	ARrStnFilterPressurePV 								: ARRAY [1..iStnQty] OF REAL;
	ARbStnFilterPressure1stLimitAlarm					: ARRAY [1..iStnQty] OF BOOL;
	ARbStnFilterPressure2ndLimitAlarm					: ARRAY [1..iStnQty] OF BOOL;

	ARbStnFilterPressureLowAlarm						: ARRAY [1..iStnQty] OF BOOL;
	ARbStnFilterPressureHighAlarm						: ARRAY [1..iStnQty] OF BOOL;
	
	ARrIncFilterPressurePV 								: ARRAY [1..iStnQty] OF REAL;
	ARbIncFilterPressure1stLimitAlarm					: ARRAY [1..iStnQty] OF BOOL;
	ARbIncFilterPressure2ndLimitAlarm					: ARRAY [1..iStnQty] OF BOOL;

(* xxxxxxxxxxxxxxxxxxxxxxxxxxxxxxxx Flow Switch Cltr xxxxxxxxxxxxxxxxxxxxxxxxxxxxxxxx*)
(*========================================================================*)

	ARrStnFlowSwitchPV 									: ARRAY [1..iStnQty] OF REAL;
	ARbStnFlowSwitch1stLimitAlarm						: ARRAY [1..iStnQty] OF BOOL;
	ARbStnFlowSwitch2ndLimitAlarm						: ARRAY [1..iStnQty] OF BOOL;

	ARrIncFlowSwitchPV 									: ARRAY [1..iStnQty] OF REAL;
	ARbIncFlowSwitch1stLimitAlarm						: ARRAY [1..iStnQty] OF BOOL;
	ARbIncFlowSwitch2ndLimitAlarm						: ARRAY [1..iStnQty] OF BOOL;

(* xxxxxxxxxxxxxxxxxxxxxxxxxxxxxxxx Compress Air Cltr xxxxxxxxxxxxxxxxxxxxxxxxxxxxxxxx*)
(*========================================================================*)

	ARrStnCompressAirPV 								: ARRAY [1..iStnQty] OF REAL;
	ARbStnCompressAir1stLimitAlarm						: ARRAY [1..iStnQty] OF BOOL;
	ARbStnCompressAir2ndLimitAlarm						: ARRAY [1..iStnQty] OF BOOL;

	ARrIncCompressAirPV 								: ARRAY [1..iStnQty] OF REAL;
	ARbIncCompressAir1stLimitAlarm						: ARRAY [1..iStnQty] OF BOOL;
	ARbIncCompressAir2ndLimitAlarm						: ARRAY [1..iStnQty] OF BOOL;

(* xxxxxxxxxxxxxxxxxxxxxxxxxxxxxx Weber Ultrasonic Cltr xxxxxxxxxxxxxxxxxxxxxxxxxxxxxx*)
(*========================================================================*)

	bWeberFbErrorReset 									: BOOL;

	ARbUSFSel1OnOff 									: ARRAY [1..iUSGeneratorQty] OF BOOL;
	ARbUSFSel2OnOff 									: ARRAY [1..iUSGeneratorQty] OF BOOL;

(* xxxxxxxxxxxxxxxxxxxxxxxxxxxxxx Brenson Ultrasonic Cltr xxxxxxxxxxxxxxxxxxxxxxxxxxxxxx*)
(*========================================================================*)

	bBrensonFbErrorReset 								: BOOL;

	ARbBrensonUSFSel1OnOff 								: ARRAY [1..iUSGeneratorQty] OF BOOL;
	ARbBrensonUSFSel2OnOff 								: ARRAY [1..iUSGeneratorQty] OF BOOL;

(* xxxxxxxxxxxxxxxxxxxxxx Manual WeberUltrasonic Variable Cltr xxxxxxxxxxxxxxxxxxxxxx*)
(*========================================================================*)

	ARiStnUSSideAPv									: ARRAY [1..iStnQty] OF INT;
	ARiStnUSSideBPv									: ARRAY [1..iStnQty] OF INT;
	ARiStnUSSideCPv									: ARRAY [1..iStnQty] OF INT;
	ARiStnUSSideDPv									: ARRAY [1..iStnQty] OF INT;

	ARiStnUSBtmAPv									: ARRAY [1..iStnQty] OF INT;
	ARiStnUSBtmBPv									: ARRAY [1..iStnQty] OF INT;
	ARiStnUSBtmCPv									: ARRAY [1..iStnQty] OF INT;
	ARiStnUSBtmDPv									: ARRAY [1..iStnQty] OF INT;
	                                                
	ARiStnUSSideAFreqPv								: ARRAY [1..iStnQty] OF INT;
	ARiStnUSSideBFreqPv								: ARRAY [1..iStnQty] OF INT;
	ARiStnUSSideCFreqPv								: ARRAY [1..iStnQty] OF INT;
	ARiStnUSSideDFreqPv								: ARRAY [1..iStnQty] OF INT;

	ARiStnUSBtmAFreqPv								: ARRAY [1..iStnQty] OF INT;
	ARiStnUSBtmBFreqPv								: ARRAY [1..iStnQty] OF INT;
	ARiStnUSBtmCFreqPv								: ARRAY [1..iStnQty] OF INT;
	ARiStnUSBtmDFreqPv								: ARRAY [1..iStnQty] OF INT;

(* xxxxxxxxxxxxxxxxxxxxxx ClangsonicUltrasonic Variable Cltr xxxxxxxxxxxxxxxxxxxxxx*)
(*========================================================================*)

	ARiUsPowerPV_percent								: ARRAY [1..12] OF INT;
	ARiUsOutput_Watt										: ARRAY [1..12] OF INT;

	ARbUSfeedbackInRange								: ARRAY [1..12] OF BOOL;

(* xxxxxxxxxxxxxxxxxxxxxxxxxxxxxxxx Inverter Encoder Cltr xxxxxxxxxxxxxxxxxxxxxxxxxxxxxxxx*)
(*========================================================================*)

	ARbVertCounterValueReset 							: ARRAY [0..iArmQty] OF BOOL;
	ARbHorzCounterValueReset 							: ARRAY [0..iArmQty] OF BOOL;

	ARbVertCounterValueErrReset 							: ARRAY [0..iArmQty] OF BOOL;
	ARbHorzCounterValueErrReset							: ARRAY [0..iArmQty] OF BOOL;

	ARbVertCounterValueErr								: ARRAY [0..iArmQty] OF BOOL;
	ARbHorzCounterValueErr								: ARRAY [0..iArmQty] OF BOOL;

	ARbVertOUT_CounterResetEn							: ARRAY [0..iArmQty] OF BOOL;
	ARbHorzOUT_CounterResetEn							: ARRAY [0..iArmQty] OF BOOL;

(* xxxxxxxxxxxxxxxxxxxxxxxxxxxxxxxx Vacuum Value Cltr xxxxxxxxxxxxxxxxxxxxxxxxxxxxxxxx*)
(*========================================================================*)

	ARbStnHighVacuumSignal								: ARRAY [1..iStnQty] OF BOOL;
	ARbStnLowVacuumSignal								: ARRAY [1..iStnQty] OF BOOL;

	ARbStnSubHighVacuumSignal							: ARRAY [1..iStnQty] OF BOOL;
	ARbStnSubLowVacuumSignal							: ARRAY [1..iStnQty] OF BOOL;

	bDCHighVacuumSignal								: BOOL;
	bDCLowVacuumSignal									: BOOL;

	bCCHighVacuumSignal								: BOOL;
	bCCLowVacuumSignal									: BOOL;

	ARbRevHighVacuumSignal								: ARRAY [1..iStnQty] OF BOOL;
	ARbRevLowVacuumSignal								: ARRAY [1..iStnQty] OF BOOL;

	ARrStnVacuumPV										: ARRAY [1..iStnQty] OF REAL;
	ARiStnVacuumPV										: ARRAY [1..iStnQty] OF INT;

	ARrStnSubVacuumPV									: ARRAY [1..iStnQty] OF REAL;
	ARiStnSubVacuumPV									: ARRAY [1..iStnQty] OF INT;

	rDCVacuumPV										: REAL;
	iDCVacuumPV										: INT;

	rCCVacuumPV										: REAL;
	iCCVacuumPV										: INT;

	ARrRevVacuumPV									: ARRAY [1..iStnQty] OF REAL;
	ARiRevVacuumPV									: ARRAY [1..iStnQty] OF INT;

	ARtVacuumPumpTimerResetDelay 						: ARRAY [1..iStnQty] OF TON;

	ARbVacuumPumpTimerReset							: ARRAY [1..iStnQty] OF BOOL;

	ARbDaysPvReset_Routine								: ARRAY [1..iStnQty] OF BOOL;
	ARbDaysPvReset_Major								: ARRAY [1..iStnQty] OF BOOL;

	ARbVacuumWarning_Routine							: ARRAY [1..iStnQty] OF BOOL;
	ARbVacuumAlarm_Routine								: ARRAY [1..iStnQty] OF BOOL;

	ARbVacuumWarning_Major								: ARRAY [1..iStnQty] OF BOOL;
	ARbVacuumAlarm_Major								: ARRAY [1..iStnQty] OF BOOL;

	ARbVacPumpService1stLimitAlarm						: ARRAY [1..iStnQty] OF BOOL;
	ARbVacPumpService2ndLimitAlarm						: ARRAY [1..iStnQty] OF BOOL;
	ARbVacPumpService2ndlimitAlarmHR					: ARRAY [1..iStnQty] OF BOOL;

(* xxxxxxxxxxxxxxxxxxxxxxxxxxx Keyence Vacuum Variable Cltr xxxxxxxxxxxxxxxxxxxxxxxxxxx*)
(*========================================================================*)

	ARbStnHighVacuumLvlSave							: ARRAY [1..iStnQty] OF BOOL;
	ARbStnLowVacuumLvlSave							: ARRAY [1..iStnQty] OF BOOL;

	ARbStnSubHighVacuumLvlSave						: ARRAY [1..iStnQty] OF BOOL;
	ARbStnSubLowVacuumLvlSave							: ARRAY [1..iStnQty] OF BOOL;

	bDCHighVacuumLvlSave								: BOOL;
	bDCLowVacuumLvlSave								: BOOL;

	bCCHighVacuumLvlSave								: BOOL;
	bCCLowVacuumLvlSave								: BOOL;

	ARbRevHighVacuumLvlSave							: ARRAY [1..iStnQty] OF BOOL;
	ARbRevLowVacuumLvlSave							: ARRAY [1..iStnQty] OF BOOL;

END_VAR

// ---- GVLs/Analog_Ctrl/Global_Variables_Analog_Persistent.TcGVL
{attribute 'Tc2GvlVarNames'}
VAR_GLOBAL PERSISTENT

(* xxxxxxxxxxxxxxxxxxxxxxxxxxxxxxxx Temperature Cltr xxxxxxxxxxxxxxxxxxxxxxxxxxxxxxxx*)
(*========================================================================*)

	ARfbStnTempControl									: ARRAY [1..iStnQty] OF fbV2_TempControl;

	ARrAnalogInputFineTuneRatio							: ARRAY [1..iStnQty] OF REAL;

	ARrStnTempHYSsv										: ARRAY [1..iStnQty] OF REAL;
	ARrStnTempHALsv										: ARRAY [1..iStnQty] OF REAL;
	ARrStnTempSV										: ARRAY [1..iStnQty] OF REAL;
	ARrStnTempRDYsv										: ARRAY [1..iStnQty] OF REAL;
	ARrStnTemp1stLimitSv								: ARRAY [1..iStnQty] OF REAL;
	ARrStnTemp2ndLimitSv								: ARRAY [1..iStnQty] OF REAL;
	ARiStnPreparationTempSv								: ARRAY [1..iStnQty] OF INT;
	
	ARrStnTempHYSMINsv									: ARRAY [1..iStnQty] OF REAL;
	ARrStnTempHYSMAXsv									: ARRAY [1..iStnQty] OF REAL;
	
	ARrStnTempHALMINsv									: ARRAY [1..iStnQty] OF REAL;
	ARrStnTempHALMAXsv									: ARRAY [1..iStnQty] OF REAL;
	
	ARrStnTempMINsv										: ARRAY [1..iStnQty] OF REAL;
	ARrStnTempMAXsv										: ARRAY [1..iStnQty] OF REAL;
	
	ARrStnTempRDYMINsv									: ARRAY [1..iStnQty] OF REAL;
	ARrStnTempRDYMAXsv									: ARRAY [1..iStnQty] OF REAL;
	
	ARrStnTemp1stLimitMINsv								: ARRAY [1..iStnQty] OF REAL;
	ARrStnTemp1stLimitMAXsv								: ARRAY [1..iStnQty] OF REAL;
	
	ARiStnPreparationTempMINsv							: ARRAY [1..iStnQty] OF INT;
	ARiStnPreparationTempMAXsv							: ARRAY [1..iStnQty] OF INT;
	
	fbChillerSystemTempControl							: fbV2_TempControl;
	
	rChillerSystemAnalogInputFineTuneRatio				: REAL;

	rChillerSystemTempHYSsv								: REAL;
	rChillerSystemTempHALsv								: REAL;
	rChillerSystemTempSV								: REAL;
	rChillerSystemTempRDYsv								: REAL;
	rChillerSystemTemp1stLimitSv						: REAL;
	rChillerSystemTemp2ndLimitSv						: REAL;
	iChillerSystemPreparationTempSv						: INT;
	
		rChillerSystemTempHYSMINsv							: REAL;
	rChillerSystemTempHYSMAXsv							: REAL;
	
	rChillerSystemTempHALMINsv							: REAL;
	rChillerSystemTempHALMAXsv							: REAL;
	
	rChillerSystemTempMINsv								: REAL;
	rChillerSystemTempMAXsv								: REAL;
	
	rChillerSystemTempRDYMINsv							: REAL;
	rChillerSystemTempRDYMAXsv							: REAL;
	
	rChillerSystemTemp1stLimitMINsv						: REAL;
	rChillerSystemTemp1stLimitMAXsv						: REAL;
	
	iChillerSystemPreparationTempMINsv					: INT;
	iChillerSystemPreparationTempMAXsv					: INT;
	

	ARrStnChillerValueTempSetpoint						: ARRAY [1..iStnQty] OF REAL;
	
		rChillerSystemTempMINsvHMIDisplay					: REAL;
	rChillerSystemTempMAXsvHMIDisplay					: REAL;
	
	rChillerSystemTempHALMINsvHMIDisplay				: REAL;
	rChillerSystemTempHALMAXsvHMIDisplay				: REAL;
	
	rChillerSystemTempHYSMINsvHMIDisplay				: REAL;
	rChillerSystemTempHYSMAXsvHMIDisplay				: REAL;
	
	rChillerSystemTempRDYMINsvHMIDisplay				: REAL;
	rChillerSystemTempRDYMAXsvHMIDisplay				: REAL;
	
	rChillerSystemTemp1stLimitMINsvHMIDisplay			: REAL;
	rChillerSystemTemp1stLimitMAXsvHMIDisplay			: REAL;
	
	iChillerSystemPreparationTempMINsvHMIDisplay		: INT;
	iChillerSystemPreparationTempMAXsvHMIDisplay		: INT;

(*****Temperature Changed Based on Recipe Ctrl *****)

	fbTemperatureParaRecipe								: fbV3_TemperatureParaRecipe;

	DSTempCtrlParameter_Min 							: DSV3_TempCtrlParameter;
	DSTempCtrlParameter_Max 							: DSV3_TempCtrlParameter;

	HMI_DSTempCtrlParameter_Input 						: DSV3_TempCtrlParameter;

(* xxxxxxxxxxxxxxxxxxxxxxxxxxxxxxxx Conductivity Cltr xxxxxxxxxxxxxxxxxxxxxxxxxxxxxxxx*)
(*========================================================================*)

	ARfbStnConductivity 									: ARRAY [1..iStnQty] OF fbRawRatioConversionReal;

	ARrStnLowConductivitySv									: ARRAY [1..iStnQty] OF REAL;
	ARrStnHighConductivitySv								: ARRAY [1..iStnQty] OF REAL;
	ARrStnConductivity1stLimitSv							: ARRAY [1..iStnQty] OF REAL;
	ARrStnConductivity2ndLimitSv							: ARRAY [1..iStnQty] OF REAL;

	bStnConductivityMaxLimitReach							: ARRAY [1..iStnQty] OF BOOL;
	ARsConductivityMsgStatus								: ARRAY [1..iStnQty] OF STRING;

(* xxxxxxxxxxxxxxxxxxxxxxxxxxxxxxxx Resistivity Cltr xxxxxxxxxxxxxxxxxxxxxxxxxxxxxxxx*)
(*========================================================================*)

	ARfbStnResistivity 										: ARRAY [1..iStnQty] OF fbRawRatioConversionReal;
                                                	
	ARrStnLowResistivitySv									: ARRAY [1..iStnQty] OF REAL;
	ARrStnHighResistivitySv									: ARRAY [1..iStnQty] OF REAL;
	ARrStnResistivity1stLimitSv									: ARRAY [1..iStnQty] OF REAL;
	ARrStnResistivity2ndLimitSv								: ARRAY [1..iStnQty] OF REAL;

	fbIncResistivity										: fbRawRatioConversionReal;
	rIncLowResistivitySv									: REAL;
	rIncHighResistivitySv									: REAL;
	rIncResistivity1stLimitSv								: REAL;
	rIncResistivity2ndLimitSv								: REAL;

(* xxxxxxxxxxxxxxxxxxxxxxxxxxxxxxxx PH Cltr xxxxxxxxxxxxxxxxxxxxxxxxxxxxxxxx*)
(*========================================================================*)

	ARfbStnPH 											: ARRAY [1..iStnQty] OF fbRawRatioConversionReal;

	ARrStnLowPHSv										: ARRAY [1..iStnQty] OF REAL;
	ARrStnHighPHSv										: ARRAY [1..iStnQty] OF REAL;
	ARrStnPH1stLimitSv									: ARRAY [1..iStnQty] OF REAL;
	ARrStnPH2ndLimitSv									: ARRAY [1..iStnQty] OF REAL;

(* xxxxxxxxxxxxxxxxxxxxxxxxxxxxxxxx Filter Pressure Cltr xxxxxxxxxxxxxxxxxxxxxxxxxxxxxxxx*)
(*========================================================================*)

	ARfbStnFilterPressure 									: ARRAY [1..iStnQty] OF fbRawRatioConversionReal;

	ARrStnLowFilterPressureSv								: ARRAY [1..iStnQty] OF REAL;
	ARrStnHighFilterPressureSv								: ARRAY [1..iStnQty] OF REAL;
	ARrStnFilterPressure1stLimitSv							: ARRAY [1..iStnQty] OF REAL;
	ARrStnFilterPressure2ndLimitSv							: ARRAY [1..iStnQty] OF REAL;

	ARfbIncFilterPressure									: ARRAY [1..iStnQty] OF fbRawRatioConversionReal;
	ARrIncLowFilterPressureSv								: ARRAY [1..iStnQty] OF REAL;
	ARrIncHighFilterPressureSv								: ARRAY [1..iStnQty] OF REAL;
	ARrIncFilterPressure1stLimitSv							: ARRAY [1..iStnQty] OF REAL;
	ARrIncFilterPressure2ndLimitSv							: ARRAY [1..iStnQty] OF REAL;

(* xxxxxxxxxxxxxxxxxxxxxxxxxxxxxxxx Flow Switch Cltr xxxxxxxxxxxxxxxxxxxxxxxxxxxxxxxx*)
(*========================================================================*)

	ARfbStnFlowSwitch 									: ARRAY [1..iStnQty] OF fbRawRatioConversionReal;

	ARrStnLowFlowSwitchSv								: ARRAY [1..iStnQty] OF REAL;
	ARrStnHighFlowSwitchSv								: ARRAY [1..iStnQty] OF REAL;
	ARrStnFlowSwitch1stLimitSv							: ARRAY [1..iStnQty] OF REAL;
	ARrStnFlowSwitch2ndLimitSv							: ARRAY [1..iStnQty] OF REAL;

	ARfbIncFlowSwitch									: ARRAY [1..iStnQty] OF fbRawRatioConversionReal;
	ARrIncLowFlowSwitchSv								: ARRAY [1..iStnQty] OF REAL;
	ARrIncHighFlowSwitchSv								: ARRAY [1..iStnQty] OF REAL;
	ARrIncFlowSwitch1stLimitSv							: ARRAY [1..iStnQty] OF REAL;
	ARrIncFlowSwitch2ndLimitSv							: ARRAY [1..iStnQty] OF REAL;

(* xxxxxxxxxxxxxxxxxxxxxxxxxxxxxxxx Compress Air Cltr xxxxxxxxxxxxxxxxxxxxxxxxxxxxxxxx*)
(*========================================================================*)

	ARfbStnCompressAir 									: ARRAY [1..iStnQty] OF fbRawRatioConversionReal;

	ARrStnLowCompressAirSv								: ARRAY [1..iStnQty] OF REAL;
	ARrStnHighCompressAirSv								: ARRAY [1..iStnQty] OF REAL;
	ARrStnCompressAir1stLimitSv							: ARRAY [1..iStnQty] OF REAL;
	ARrStnCompressAir2ndLimitSv							: ARRAY [1..iStnQty] OF REAL;

	ARfbIncCompressAir									: ARRAY [1..iStnQty] OF fbRawRatioConversionReal;
	ARrIncLowCompressAirSv								: ARRAY [1..iStnQty] OF REAL;
	ARrIncHighCompressAirSv								: ARRAY [1..iStnQty] OF REAL;
	ARrIncCompressAir1stLimitSv							: ARRAY [1..iStnQty] OF REAL;
	ARrIncCompressAir2ndLimitSv							: ARRAY [1..iStnQty] OF REAL;

(* xxxxxxxxxxxxxxxxxxxxxx Manual WeberUltrasonic Variable Cltr xxxxxxxxxxxxxxxxxxxxxx*)
(*========================================================================*)

	ARiStnManualUSSideAsv								: ARRAY [1..iStnQty] OF INT;
	ARiStnManualUSSideBsv								: ARRAY [1..iStnQty] OF INT;
	ARiStnManualUSSideCsv								: ARRAY [1..iStnQty] OF INT;
	ARiStnManualUSSideDsv								: ARRAY [1..iStnQty] OF INT;

	ARiStnManualUSBtmAsv								: ARRAY [1..iStnQty] OF INT;
	ARiStnManualUSBtmBsv								: ARRAY [1..iStnQty] OF INT;
	ARiStnManualUSBtmCsv								: ARRAY [1..iStnQty] OF INT;
	ARiStnManualUSBtmDsv								: ARRAY [1..iStnQty] OF INT;

(* xxxxxxxxxxxxxxxxxxxxxx Blower Inverter Variable Cltr xxxxxxxxxxxxxxxxxxxxxx*)
(*========================================================================*)

	ARiStnManualBlowerInvPercentSV						: ARRAY [1..iStnQty] OF INT;

(* xxxxxxxxxxxxxxxxxxxxxxxxxxxx Clangsonic Ultrasonic Cltr xxxxxxxxxxxxxxxxxxxxxxxxxxxx*)
(*========================================================================*)

	DSClangGenerator 									: ARRAY [1..iUSGeneratorQty] OF DS_ClangsonicGenerator;
	DSClangGenerator2 									: ARRAY [1..iUSGeneratorQty] OF DS_ClangsonicGenerator;
	iClangStepDelaySVns									: INT := 50;
	iClangStepDelaySVns2								: INT := 50;

	iClangTolerance										: INT;
	iUSTolerance										: INT;
	ARlrUsMaxData_Watt									: ARRAY [1..12] OF LREAL;

	DSClangsonicGenerator 								: DSV2_ClangsonicGenerator;
	DSClangsonicGenerator2 								: DSV2_ClangsonicGenerator;

(* xxxxxxxxxxxxxxxxxxxxxxxxxxxxxxxx Inverter Encoder Cltr xxxxxxxxxxxxxxxxxxxxxxxxxxxxxxxx*)
(*========================================================================*)

	ARlrVertRatioPulseToMM 								: ARRAY [0..iArmQty] OF LREAL;
	ARlrHorzRatioPulseToMM 								: ARRAY [0..iArmQty] OF LREAL;

	ARiVertCounterValueResetTime_Sec 					: ARRAY [0..iArmQty] OF INT;
	ARiHorzCounterValueResetTime_Sec 					: ARRAY [0..iArmQty] OF INT;

	ARrVertGen_In_HzToRawRatio							: ARRAY [0..iArmQty] OF REAL ;
	ARrHorzGen_In_HzToRawRatio							: ARRAY [0..iArmQty] OF REAL ;

(* xxxxxxxxxxxxxxxxxxxxxxxxxxxxxxxx Vacuum Value Cltr xxxxxxxxxxxxxxxxxxxxxxxxxxxxxxxx*)
(*========================================================================*)

	ARrStnHighVacuumLevelSV							: ARRAY [1..iStnQty] OF REAL;
	ARrStnLowVacuumLevelSV								: ARRAY [1..iStnQty] OF REAL;

	ARrStnSubHighVacuumLevelSV							: ARRAY [1..iStnQty] OF REAL;
	ARrStnSubLowVacuumLevelSV							: ARRAY [1..iStnQty] OF REAL;

	rDCHighVacuumLevelSV								: REAL;
	rDCLowVacuumLevelSV								: REAL;

	rJRSCCHighVacuumLevelSV							: REAL;
	rJRSCCLowVacuumLevelSV							: REAL;

	ARrCCHighVacuumLevelSV							: ARRAY [1..iStnQty] OF REAL;
	ARrCCLowVacuumLevelSV								: ARRAY [1..iStnQty] OF REAL;

	ARrRevHighVacuumLevelSV							: ARRAY [1..iStnQty] OF REAL;
	ARrRevLowVacuumLevelSV							: ARRAY [1..iStnQty] OF REAL;

	ARdiVacPump1stLimitTimerSV							: ARRAY [1..iStnQty] OF DINT;
	ARdiVacPump2ndLimitTimerSV							: ARRAY [1..iStnQty] OF DINT;

	ARiWarningDaysSV_Routine							: ARRAY [1..iStnQty] OF INT;
	ARiAlarmDaysSV_Routine								: ARRAY [1..iStnQty] OF INT;

	ARiRunDaysPV_Routine								: ARRAY [1..iStnQty] OF INT;
	ARsPreviousDate_Routine								: ARRAY [1..iStnQty] OF STRING;

	ARiWarningDaysSV_Major								: ARRAY [1..iStnQty] OF INT;
	ARiAlarmDaysSV_Major								: ARRAY [1..iStnQty] OF INT;

	ARiRunDaysPV_Major									: ARRAY [1..iStnQty] OF INT;
	ARsPreviousDate_Major								: ARRAY [1..iStnQty] OF STRING;

(* xxxxxxxxxxxxxxxxxxxxxxxxxxx Keyence Vacuum Variable Cltr xxxxxxxxxxxxxxxxxxxxxxxxxxx*)
(*========================================================================*)

	fbDCVacuumSensorCtrl								: fbKeyenceVacSensorTuningkPa;
	fbJRSCCVacuumSensorCtrl								: fbKeyenceVacSensorTuningkPa;
	ARfbCCVacuumSensorCtrl								: ARRAY [1..iStnQty] OF fbKeyenceVacSensorTuningkPa;
	ARfbStnVacuumSensorCtrl								: ARRAY [1..iStnQty] OF fbKeyenceVacSensorTuningkPa;
	ARfbStnSubVacuumSensorCtrl							: ARRAY [1..iStnQty] OF fbKeyenceVacSensorTuningkPa;
	ARfbRevVacuumSensorCtrl								: ARRAY [1..iStnQty] OF fbKeyenceVacSensorTuningkPa;

	ARlrStnVacuumMaxReadSV							: ARRAY [1..iStnQty] OF LREAL;
	ARlrStnSubVacuumMaxReadSV							: ARRAY [1..iStnQty] OF LREAL;

	lrDCVacuumMaxReadSV								: LREAL;
	lrJRSCCVacuumMaxReadSV							: LREAL;
	ARlrCCVacuumMaxReadSV							: ARRAY [1..iStnQty] OF LREAL;
	ARlrRevVacuumMaxReadSV							: ARRAY [1..iStnQty] OF LREAL;
	
(* xxxxxxxxxxxxxxxxxxxxxxxxxxx Modbus Cltr xxxxxxxxxxxxxxxxxxxxxxxxxxx*)
(*========================================================================*)
	DSV2ModbusControl									: DSV2_ModbusControl;
	DSV2ModbusControl2 									: DSV2_ModbusControl;
	
	IStepDelaySVns										: INT := 50;
	IStepDelaySVns2										: INT := 50;


END_VAR

// ---- GVLs/Analog_Ctrl/Global_Variables_DeclarationOnly.TcGVL
{attribute 'Tc2GvlVarNames'}
VAR_GLOBAL

(* xxxxxxxxxxxxxxxxxxxxxxxxxxxxxx Weber Ultrasonic Cltr xxxxxxxxxxxxxxxxxxxxxxxxxxxxxx*)
(*========================================================================*)

	DSWeberGenerator 									: ARRAY [1..iUSGeneratorQty] OF DS_WeberGenerator;
	DSWeberEnclosure 									: ARRAY [1..iUSEnclosureQty] OF DS_WeberEnclosure;
	iWeberStepDelaySVns									: INT;

	ARfbWeberMultiFreq_Main								: ARRAY [1..4] OF fbWeberMultiFreqCtrl;

(* xxxxxxxxxxxxxxxxxxxxxxxxxxxxxx Brenson Ultrasonic Cltr xxxxxxxxxxxxxxxxxxxxxxxxxxxxxx*)
(*========================================================================*)

	DSBrensonGenerator 									: ARRAY [1..iUSGeneratorQty] OF DS_BrensonGenerator;
	DSBrensonEnclosure 									: ARRAY [1..iUSEnclosureQty] OF DS_BrensonEnclosure;
	iBrensonStepDelaySVns								: INT;

	ARfbBrensonMultiFreq_Main							: ARRAY [1..4] OF fbBrensonMultiFreqCtrl;

(* xxxxxxxxxxxxxxxxxxxxxxxxxxxx Clangsonic Ultrasonic Cltr xxxxxxxxxxxxxxxxxxxxxxxxxxxx*)
(*========================================================================*)

	bClang_ModbusReadBusy								: BOOL;
	bClang_ModbusReadError								: BOOL;
	bClang_ModbusWriteBusy								: BOOL;
	bClang_ModbusWriteError								: BOOL;

	ErrorId_Read										: MODBUS_ERRORS;
	ErrorId_Write										: MODBUS_ERRORS;

	bClang_ModbusReadBusy2								: BOOL;
	bClang_ModbusReadError2								: BOOL;
	bClang_ModbusWriteBusy2								: BOOL;
	bClang_ModbusWriteError2							: BOOL;

	ErrorId_Read2										: MODBUS_ERRORS;
	ErrorId_Write2										: MODBUS_ERRORS;
	
(* xxxxxxxxxxxxxxxxxxxxxxxxxxxx Generic  Modbus Cltr xxxxxxxxxxxxxxxxxxxxxxxxxxxx*)
(*========================================================================*)
	
	bModbusReadBusy										: BOOL;
	bModbusReadError									: BOOL;
	bModbusWriteBusy									: BOOL;
	bModbusWriteError									: BOOL;
	
	bModbusReadBusy2									: BOOL;
	bModbusReadError2									: BOOL;
	bModbusWriteBusy2									: BOOL;
	bModbusWriteError2									: BOOL;

END_VAR

// ---- GVLs/Arm_Ctrl/Global_Variables_Arm1BoolCtrl.TcGVL
{attribute 'Tc2GvlVarNames'}
VAR_GLOBAL

(*HORZ*)

	dwArm1HorzHomeStart 		: DWORD; (* %MD20900 *)
	dwArm1HorzHomeReset 		: DWORD; (* %MD20940 *)

(* xxx Horz SlantedLeft DWORD LINK with %MX20000-MX20099  xxx*)
(*======================================================*)

	dwArm1HorzStn1SlantedLeft 	: DWORD; (* %MD20004 *)
	dwArm1HorzStn2SlantedLeft 	: DWORD; (* %MD20008 *)
	dwArm1HorzStn3SlantedLeft 	: DWORD; (* %MD20012 *)
	dwArm1HorzStn4SlantedLeft 	: DWORD; (* %MD20016 *)
	dwArm1HorzStn5SlantedLeft 	: DWORD; (* %MD20020 *)
	dwArm1HorzStn6SlantedLeft 	: DWORD; (* %MD20024 *)
	dwArm1HorzStn7SlantedLeft 	: DWORD; (* %MD20028 *)
	dwArm1HorzStn8SlantedLeft 	: DWORD; (* %MD20032 *)
	dwArm1HorzStn9SlantedLeft 	: DWORD; (* %MD20036 *)
	dwArm1HorzStn10SlantedLeft 	: DWORD; (* %MD20040 *)
	dwArm1HorzStn11SlantedLeft 	: DWORD; (* %MD20044 *)
	dwArm1HorzStn12SlantedLeft 	: DWORD; (* %MD20048 *)

(* xxx Horz SlantedRight DWORD LINK with %MX20100-MX20199  xxx*)
(*======================================================*)

	dwArm1HorzStn1SlantedRight 	: DWORD; (* %MD20104 *)
	dwArm1HorzStn2SlantedRight	: DWORD; (* %MD20108 *)
	dwArm1HorzStn3SlantedRight 	: DWORD; (* %MD20112 *)
	dwArm1HorzStn4SlantedRight	: DWORD; (* %MD20116 *)
	dwArm1HorzStn5SlantedRight 	: DWORD; (* %MD20120 *)
	dwArm1HorzStn6SlantedRight 	: DWORD; (* %MD20124 *)
	dwArm1HorzStn7SlantedRight 	: DWORD; (* %MD20128 *)
	dwArm1HorzStn8SlantedRight 	: DWORD; (* %MD20132 *)
	dwArm1HorzStn9SlantedRight 	: DWORD; (* %MD20136 *)
	dwArm1HorzStn10SlantedRight 	: DWORD; (* %MD20140 *)
	dwArm1HorzStn11SlantedRight 	: DWORD; (* %MD20144 *)
	dwArm1HorzStn12SlantedRight 	: DWORD; (* %MD20148 *)

(* xxx Hook DWORD LINK with %MX20200-MX20299  xxx*)
(*======================================================*)

	dwArm1Ld1Hook 				: DWORD; (* %MD20252 *)
	dwArm1Uld1Hook 			: DWORD; (* %MD20256 *)
	dwArm1HorzStn1Hook 			: DWORD; (* %MD20204 *)
	dwArm1HorzStn2Hook			: DWORD; (* %MD20208 *)
	dwArm1HorzStn3Hook 			: DWORD; (* %MD20212 *)
	dwArm1HorzStn4Hook 			: DWORD; (* %MD20216 *)
	dwArm1HorzStn5Hook 			: DWORD; (* %MD20220 *)
	dwArm1HorzStn6Hook 			: DWORD; (* %MD20224 *)
	dwArm1HorzStn7Hook 			: DWORD; (* %MD20228 *)
	dwArm1HorzStn8Hook 			: DWORD; (* %MD20232 *)
	dwArm1HorzStn9Hook 			: DWORD; (* %MD20236 *)
	dwArm1HorzStn10Hook 		: DWORD; (* %MD20240 *)
	dwArm1HorzStn11Hook 		: DWORD; (* %MD20244 *)
	dwArm1HorzStn12Hook 		: DWORD; (* %MD20248 *)

(* xxx Unhook DWORD LINK with %MX20300-MX20399  xxx*)
(*======================================================*)

	dwArm1Ld1Unhook 			: DWORD; (* %MD20352 *)
	dwArm1Uld1Unhook 			: DWORD; (* %MD20356 *)
	dwArm1HorzStn1Unhook 		: DWORD; (* %MD20304 *)
	dwArm1HorzStn2Unhook 		: DWORD; (* %MD20308 *)
	dwArm1HorzStn3Unhook 		: DWORD; (* %MD20312 *)
	dwArm1HorzStn4Unhook 		: DWORD; (* %MD20316 *)
	dwArm1HorzStn5Unhook 		: DWORD; (* %MD20320 *)
	dwArm1HorzStn6Unhook 		: DWORD; (* %MD20324 *)
	dwArm1HorzStn7Unhook 		: DWORD; (* %MD20328 *)
	dwArm1HorzStn8Unhook 		: DWORD; (* %MD20332 *)
	dwArm1HorzStn9Unhook 		: DWORD; (* %MD20336 *)
	dwArm1HorzStn10Unhook 		: DWORD; (* %MD20340 *)
	dwArm1HorzStn11Unhook 		: DWORD; (* %MD20344 *)
	dwArm1HorzStn12Unhook 		: DWORD; (* %MD20348 *)

(*VERT*)

	dwArm1VertHomeStart 			: DWORD; (* %MD25900 *)
	dwArm1VertHomeReset 		: DWORD; (* %MD25940 *)

(* xxx Up DWORD LINK with %MX25000-MX25099  xxx*)
(*======================================================*)

	dwArm1Ld1Up 				: DWORD; (* %MD25052 *)
	dwArm1Uld1Up 				: DWORD; (* %MD25056 *)
	dwArm1VertStn1Up 			: DWORD; (* %MD25004 *)
	dwArm1VertStn2Up 			: DWORD; (* %MD25008 *)
	dwArm1VertStn3Up 			: DWORD; (* %MD25012 *)
	dwArm1VertStn4Up 			: DWORD; (* %MD25016 *)
	dwArm1VertStn5Up 			: DWORD; (* %MD25020 *)
	dwArm1VertStn6Up 			: DWORD; (* %MD25024 *)
	dwArm1VertStn7Up 			: DWORD; (* %MD25028 *)
	dwArm1VertStn8Up 			: DWORD; (* %MD25032 *)
	dwArm1VertStn9Up 			: DWORD; (* %MD25036 *)
	dwArm1VertStn10Up 			: DWORD; (* %MD25040 *)
	dwArm1VertStn11Up 			: DWORD; (* %MD25044 *)
	dwArm1VertStn12Up 			: DWORD; (* %MD25048 *)

(* xxx Down SpSlanted DWORD LINK with %MX25100-MX25199  xxx*)
(*======================================================*)
(*Arm Mid Pos*)
	dwArm1VertStn1SpSlanted 		: DWORD; (* %MD25104 *)
	dwArm1VertStn2SpSlanted 		: DWORD; (* %MD25108 *)
	dwArm1VertStn3SpSlanted 		: DWORD; (* %MD25112 *)
	dwArm1VertStn4SpSlanted 		: DWORD; (* %MD25116 *)
	dwArm1VertStn5SpSlanted 		: DWORD; (* %MD25120 *)
	dwArm1VertStn6SpSlanted 		: DWORD; (* %MD25124 *)
	dwArm1VertStn7SpSlanted 		: DWORD; (* %MD25128 *)
	dwArm1VertStn8SpSlanted 		: DWORD; (* %MD25132 *)
	dwArm1VertStn9SpSlanted 		: DWORD; (* %MD25136 *)
	dwArm1VertStn10SpSlanted 	: DWORD; (* %MD25140 *)
	dwArm1VertStn11SpSlanted 	: DWORD; (* %MD25144 *)
	dwArm1VertStn12SpSlanted 	: DWORD; (* %MD25148 *)

(* xxx Down Regular DWORD LINK with %MX25200-MX25299  xxx*)
(*======================================================*)

	dwArm1VertStn1Regular 		: DWORD; (* %MD25204 *)
	dwArm1VertStn2Regular 		: DWORD; (* %MD25208 *)
	dwArm1VertStn3Regular 		: DWORD; (* %MD25212 *)
	dwArm1VertStn4Regular 		: DWORD; (* %MD25216 *)
	dwArm1VertStn5Regular 		: DWORD; (* %MD25220 *)
	dwArm1VertStn6Regular 		: DWORD; (* %MD25224 *)
	dwArm1VertStn7Regular 		: DWORD; (* %MD25228 *)
	dwArm1VertStn8Regular 		: DWORD; (* %MD25232 *)
	dwArm1VertStn9Regular 		: DWORD; (* %MD25236 *)
	dwArm1VertStn10Regular 		: DWORD; (* %MD25240 *)
	dwArm1VertStn11Regular 		: DWORD; (* %MD25244 *)
	dwArm1VertStn12Regular 		: DWORD; (* %MD25248 *)

(* xxx Up AgiUp DWORD LINK with %MX25300-MX25399  xxx*)
(*======================================================*)

	dwArm1VertStn1AglUp 			: DWORD; (* %MD25304 *)
	dwArm1VertStn2AglUp 			: DWORD; (* %MD25308 *)
	dwArm1VertStn3AglUp			: DWORD; (* %MD25312 *)
	dwArm1VertStn4AglUp 			: DWORD; (* %MD25316 *)
	dwArm1VertStn5AglUp 			: DWORD; (* %MD25320 *)
	dwArm1VertStn6AglUp 			: DWORD; (* %MD25324 *)
	dwArm1VertStn7AglUp 			: DWORD; (* %MD25328 *)
	dwArm1VertStn8AglUp 			: DWORD; (* %MD25332 *)
	dwArm1VertStn9AglUp 			: DWORD; (* %MD25336 *)
	dwArm1VertStn10AglUp 		: DWORD; (* %MD25340 *)
	dwArm1VertStn11AglUp 		: DWORD; (* %MD25344 *)
	dwArm1VertStn12AglUp 		: DWORD; (* %MD25348 *)

(* xxx Down AgiDown DWORD LINK with %MX25400-MX25499  xxx*)
(*======================================================*)

	dwArm1VertStn1AglDown 		: DWORD; (* %MD25404 *)
	dwArm1VertStn2AglDown 		: DWORD; (* %MD25408 *)
	dwArm1VertStn3AglDown 		: DWORD; (* %MD25412 *)
	dwArm1VertStn4AglDown 		: DWORD; (* %MD25416 *)
	dwArm1VertStn5AglDown 		: DWORD; (* %MD25420 *)
	dwArm1VertStn6AglDown 		: DWORD; (* %MD25424 *)
	dwArm1VertStn7AglDown 		: DWORD; (* %MD25428 *)
	dwArm1VertStn8AglDown 		: DWORD; (* %MD25432 *)
	dwArm1VertStn9AglDown 		: DWORD; (* %MD25436 *)
	dwArm1VertStn10AglDown 		: DWORD; (* %MD25440 *)
	dwArm1VertStn11AglDown 		: DWORD; (* %MD25444 *)
	dwArm1VertStn12AglDown 		: DWORD; (* %MD25448 *)

(* xxx Down DWORD LINK with %MX25500-MX25599  xxx*)
(*======================================================*)

	dwArm1Ld1Down 				: DWORD; (* %MD25552 *)
	dwArm1Uld1Down 			: DWORD; (* %MD25556 *)
	dwArm1VertStn1Down 			: DWORD; (* %MD25504 *)
	dwArm1VertStn2Down 			: DWORD; (* %MD25508 *)
	dwArm1VertStn3Down 			: DWORD; (* %MD25512 *)
	dwArm1VertStn4Down 			: DWORD; (* %MD25516 *)
	dwArm1VertStn5Down 			: DWORD; (* %MD25520 *)
	dwArm1VertStn6Down 			: DWORD; (* %MD25524 *)
	dwArm1VertStn7Down 			: DWORD; (* %MD25528 *)
	dwArm1VertStn8Down 			: DWORD; (* %MD25532 *)
	dwArm1VertStn9Down 			: DWORD; (* %MD25536 *)
	dwArm1VertStn10Down 		: DWORD; (* %MD25540 *)
	dwArm1VertStn11Down 		: DWORD; (* %MD25544 *)
	dwArm1VertStn12Down 		: DWORD; (* %MD25548 *)

(*LIFTER*)

	dwSlowPull1LifterHomeStart 	: DWORD; (* %MD30900 *)
	dwSlowPull1LifterHomeReset 	: DWORD; (* %MD30940 *)

(* xxx Up/Down LifterUp DWORD LINK with %MX30000-   xxx*)
(*======================================================*)

	dwSlowPull1LifterStn1Up 		: DWORD; (* %MD30004 *)
	dwSlowPull1LifterStn2Up 		: DWORD; (* %MD30008 *)
	dwSlowPull1LifterStn3Up 		: DWORD; (* %MD30012 *)
	dwSlowPull1LifterStn4Up 		: DWORD; (* %MD30016 *)
	dwSlowPull1LifterStn5Up 		: DWORD; (* %MD30020 *)
	dwSlowPull1LifterStn6Up 		: DWORD; (* %MD30024 *)
	dwSlowPull1LifterStn7Up 		: DWORD; (* %MD30028 *)
	dwSlowPull1LifterStn8Up 		: DWORD; (* %MD30032 *)
	dwSlowPull1LifterStn9Up 		: DWORD; (* %MD30036 *)
	dwSlowPull1LifterStn10Up 		: DWORD; (* %MD30040 *)
	dwSlowPull1LifterStn11Up 		: DWORD; (* %MD30044 *)
	dwSlowPull1LifterStn12Up 		: DWORD; (* %MD30048 *)

(* xxx Up/Down LifterDown DWORD LINK with %MX30000-   xxx*)
(*======================================================*)

	dwSlowPull1LifterStn1Down 		: DWORD; (* %MD30304 *)
	dwSlowPull1LifterStn2Down 		: DWORD; (* %MD30308 *)
	dwSlowPull1LifterStn3Down 		: DWORD; (* %MD30312 *)
	dwSlowPull1LifterStn4Down 		: DWORD; (* %MD30316 *)
	dwSlowPull1LifterStn5Down 		: DWORD; (* %MD30320 *)
	dwSlowPull1LifterStn6Down 		: DWORD; (* %MD30324 *)
	dwSlowPull1LifterStn7Down 		: DWORD; (* %MD30328 *)
	dwSlowPull1LifterStn8Down 		: DWORD; (* %MD30332 *)
	dwSlowPull1LifterStn9Down 		: DWORD; (* %MD30336 *)
	dwSlowPull1LifterStn10Down 	: DWORD; (* %MD30340 *)
	dwSlowPull1LifterStn11Down 	: DWORD; (* %MD30344 *)
	dwSlowPull1LifterStn12Down 	: DWORD; (* %MD30348 *)

(* xxx Up/Down LifterAgiUp DWORD LINK with %MX30000-   xxx*)
(*======================================================*)

	dwSlowPull1LifterStn1AgiUp 	: DWORD; (* %MD30104 *)
	dwSlowPull1LifterStn2AgiUp 	: DWORD; (* %MD30108 *)
	dwSlowPull1LifterStn3AgiUp 	: DWORD; (* %MD30112 *)
	dwSlowPull1LifterStn4AgiUp 	: DWORD; (* %MD30116 *)
	dwSlowPull1LifterStn5AgiUp 	: DWORD; (* %MD30120 *)
	dwSlowPull1LifterStn6AgiUp 	: DWORD; (* %MD30124 *)
	dwSlowPull1LifterStn7AgiUp 	: DWORD; (* %MD30128 *)
	dwSlowPull1LifterStn8AgiUp 	: DWORD; (* %MD30132 *)
	dwSlowPull1LifterStn9AgiUp 	: DWORD; (* %MD30136 *)
	dwSlowPull1LifterStn10AgiUp 	: DWORD; (* %MD30140 *)
	dwSlowPull1LifterStn11AgiUp 	: DWORD; (* %MD30144 *)
	dwSlowPull1LifterStn12AgiUp 	: DWORD; (* %MD30148 *)

(* xxx Up/Down LifterAgiDown DWORD LINK with %MX30000-   xxx*)
(*======================================================*)

	dwSlowPull1LifterStn1AgiDown 	: DWORD; (* %MD30204 *)
	dwSlowPull1LifterStn2AgiDown 	: DWORD; (* %MD30208 *)
	dwSlowPull1LifterStn3AgiDown 	: DWORD; (* %MD30212 *)
	dwSlowPull1LifterStn4AgiDown 	: DWORD; (* %MD30216 *)
	dwSlowPull1LifterStn5AgiDown 	: DWORD; (* %MD30220 *)
	dwSlowPull1LifterStn6AgiDown 	: DWORD; (* %MD30224 *)
	dwSlowPull1LifterStn7AgiDown 	: DWORD; (* %MD30228 *)
	dwSlowPull1LifterStn8AgiDown 	: DWORD; (* %MD30232 *)
	dwSlowPull1LifterStn9AgiDown 	: DWORD; (* %MD30236 *)
	dwSlowPull1LifterStn10AgiDown 	: DWORD; (* %MD30240 *)
	dwSlowPull1LifterStn11AgiDown 	: DWORD; (* %MD30244 *)
	dwSlowPull1LifterStn12AgiDown 	: DWORD; (* %MD30248 *)

(* xxxxxxxxxxxxxxxxxxxxxxxxxxxxxxxxxxxxxxx Home xxxxxxxxxxxxxxxxxxxxxxxxxxxxxxxxxxxxxxx*)
(*====================== Vert Home BOOL LINK with %MX25900 ======================*)

	bArm1VertHomeStart_00 AT %MX25900.0 : BOOL;
	bArm1VertHomeStart_01 AT %MX25900.1 : BOOL;
	bArm1VertHomeStart_02 AT %MX25900.2 : BOOL;
	bArm1VertHomeStart_03 AT %MX25900.3 : BOOL;
	bArm1VertHomeStart_04 AT %MX25900.4 : BOOL;
	bArm1VertHomeStart_05 AT %MX25900.5 : BOOL;
	bArm1VertHomeStart_06 AT %MX25900.6 : BOOL;
	bArm1VertHomeStart_07 AT %MX25900.7 : BOOL;
	bArm1VertHomeStart_08 AT %MX25900.8 : BOOL;
	bArm1VertHomeStart_09 AT %MX25900.9 : BOOL;
	bArm1VertHomeStart_10 AT %MX25900.10 : BOOL;
	bArm1VertHomeStart_11 AT %MX25900.11 : BOOL;
	bArm1VertHomeStart_12 AT %MX25900.12 : BOOL;
	bArm1VertHomeStart_13 AT %MX25900.13 : BOOL;
	bArm1VertHomeStart_14 AT %MX25900.14 : BOOL;
	bArm1VertHomeStart_15 AT %MX25900.15 : BOOL;
	bArm1VertHomeStart_16 AT %MX25900.16 : BOOL;
	bArm1VertHomeStart_17 AT %MX25900.17 : BOOL;
	bArm1VertHomeStart_18 AT %MX25900.18 : BOOL;
	bArm1VertHomeStart_19 AT %MX25900.19 : BOOL;
	bArm1VertHomeStart_20 AT %MX25900.20 : BOOL;
	bArm1VertHomeStart_21 AT %MX25900.21 : BOOL;
	bArm1VertHomeStart_22 AT %MX25900.22 : BOOL;
	bArm1VertHomeStart_23 AT %MX25900.23 : BOOL;
	bArm1VertHomeStart_24 AT %MX25900.24 : BOOL;
	bArm1VertHomeStart_25 AT %MX25900.25 : BOOL;
	bArm1VertHomeStart_26 AT %MX25900.26 : BOOL;
	bArm1VertHomeStart_27 AT %MX25900.27 : BOOL;
	bArm1VertHomeStart_28 AT %MX25900.28 : BOOL;
	bArm1VertHomeStart_29 AT %MX25900.29 : BOOL;
	bArm1VertHomeStart_30 AT %MX25900.30 : BOOL;
	bArm1VertHomeStart_31 AT %MX25900.31 : BOOL;

	bArm1HorzHomeStart_00 AT %MX20900.0 : BOOL;
	bArm1HorzHomeStart_01 AT %MX20900.1 : BOOL;
	bArm1HorzHomeStart_02 AT %MX20900.2 : BOOL;
	bArm1HorzHomeStart_03 AT %MX20900.3 : BOOL;
	bArm1HorzHomeStart_04 AT %MX20900.4 : BOOL;
	bArm1HorzHomeStart_05 AT %MX20900.5 : BOOL;
	bArm1HorzHomeStart_06 AT %MX20900.6 : BOOL;
	bArm1HorzHomeStart_07 AT %MX20900.7 : BOOL;
	bArm1HorzHomeStart_08 AT %MX20900.8 : BOOL;
	bArm1HorzHomeStart_09 AT %MX20900.9 : BOOL;
	bArm1HorzHomeStart_10 AT %MX20900.10 : BOOL;
	bArm1HorzHomeStart_11 AT %MX20900.11 : BOOL;
	bArm1HorzHomeStart_12 AT %MX20900.12 : BOOL;
	bArm1HorzHomeStart_13 AT %MX20900.13 : BOOL;
	bArm1HorzHomeStart_14 AT %MX20900.14 : BOOL;
	bArm1HorzHomeStart_15 AT %MX20900.15 : BOOL;
	bArm1HorzHomeStart_16 AT %MX20900.16 : BOOL;
	bArm1HorzHomeStart_17 AT %MX20900.17 : BOOL;
	bArm1HorzHomeStart_18 AT %MX20900.18 : BOOL;
	bArm1HorzHomeStart_19 AT %MX20900.19 : BOOL;
	bArm1HorzHomeStart_20 AT %MX20900.20 : BOOL;
	bArm1HorzHomeStart_21 AT %MX20900.21 : BOOL;
	bArm1HorzHomeStart_22 AT %MX20900.22 : BOOL;
	bArm1HorzHomeStart_23 AT %MX20900.23 : BOOL;
	bArm1HorzHomeStart_24 AT %MX20900.24 : BOOL;
	bArm1HorzHomeStart_25 AT %MX20900.25 : BOOL;
	bArm1HorzHomeStart_26 AT %MX20900.26 : BOOL;
	bArm1HorzHomeStart_27 AT %MX20900.27 : BOOL;
	bArm1HorzHomeStart_28 AT %MX20900.28 : BOOL;
	bArm1HorzHomeStart_29 AT %MX20900.29 : BOOL;
	bArm1HorzHomeStart_30 AT %MX20900.30 : BOOL;
	bArm1HorzHomeStart_31 AT %MX20900.31 : BOOL;

	bSlowPull1LifterHomeStart_00 AT %MX30900.0 : BOOL;
	bSlowPull1LifterHomeStart_01 AT %MX30900.1 : BOOL;
	bSlowPull1LifterHomeStart_02 AT %MX30900.2 : BOOL;
	bSlowPull1LifterHomeStart_03 AT %MX30900.3 : BOOL;
	bSlowPull1LifterHomeStart_04 AT %MX30900.4 : BOOL;
	bSlowPull1LifterHomeStart_05 AT %MX30900.5 : BOOL;
	bSlowPull1LifterHomeStart_06 AT %MX30900.6 : BOOL;
	bSlowPull1LifterHomeStart_07 AT %MX30900.7 : BOOL;
	bSlowPull1LifterHomeStart_08 AT %MX30900.8 : BOOL;
	bSlowPull1LifterHomeStart_09 AT %MX30900.9 : BOOL;
	bSlowPull1LifterHomeStart_10 AT %MX30900.10 : BOOL;
	bSlowPull1LifterHomeStart_11 AT %MX30900.11 : BOOL;
	bSlowPull1LifterHomeStart_12 AT %MX30900.12 : BOOL;
	bSlowPull1LifterHomeStart_13 AT %MX30900.13 : BOOL;
	bSlowPull1LifterHomeStart_14 AT %MX30900.14 : BOOL;
	bSlowPull1LifterHomeStart_15 AT %MX30900.15 : BOOL;
	bSlowPull1LifterHomeStart_16 AT %MX30900.16 : BOOL;
	bSlowPull1LifterHomeStart_17 AT %MX30900.17 : BOOL;
	bSlowPull1LifterHomeStart_18 AT %MX30900.18 : BOOL;
	bSlowPull1LifterHomeStart_19 AT %MX30900.19 : BOOL;
	bSlowPull1LifterHomeStart_20 AT %MX30900.20 : BOOL;
	bSlowPull1LifterHomeStart_21 AT %MX30900.21 : BOOL;
	bSlowPull1LifterHomeStart_22 AT %MX30900.22 : BOOL;
	bSlowPull1LifterHomeStart_23 AT %MX30900.23 : BOOL;
	bSlowPull1LifterHomeStart_24 AT %MX30900.24 : BOOL;
	bSlowPull1LifterHomeStart_25 AT %MX30900.25 : BOOL;
	bSlowPull1LifterHomeStart_26 AT %MX30900.26 : BOOL;
	bSlowPull1LifterHomeStart_27 AT %MX30900.27 : BOOL;
	bSlowPull1LifterHomeStart_28 AT %MX30900.28 : BOOL;
	bSlowPull1LifterHomeStart_29 AT %MX30900.29 : BOOL;
	bSlowPull1LifterHomeStart_30 AT %MX30900.30 : BOOL;
	bSlowPull1LifterHomeStart_31 AT %MX30900.31 : BOOL;


(*=============================== SlantedLeft word ===============================*)
(*====================== SlantedLeft BOOL LINK with %MX20000-MX20099 ======================*)

	bArm1HorzStn1SlantedLeft_00 AT %MX20004.0 : BOOL;
	bArm1HorzStn1SlantedLeft_01 AT %MX20004.1 : BOOL;
	bArm1HorzStn1SlantedLeft_02 AT %MX20004.2 : BOOL;
	bArm1HorzStn1SlantedLeft_03 AT %MX20004.3 : BOOL;
	bArm1HorzStn1SlantedLeft_04 AT %MX20004.4 : BOOL;
	bArm1HorzStn1SlantedLeft_05 AT %MX20004.5 : BOOL;
	bArm1HorzStn1SlantedLeft_06 AT %MX20004.6 : BOOL;
	bArm1HorzStn1SlantedLeft_07 AT %MX20004.7 : BOOL;
	bArm1HorzStn1SlantedLeft_08 AT %MX20004.8 : BOOL;
	bArm1HorzStn1SlantedLeft_09 AT %MX20004.9 : BOOL;
	bArm1HorzStn1SlantedLeft_10 AT %MX20004.10 : BOOL;
	bArm1HorzStn1SlantedLeft_11 AT %MX20004.11 : BOOL;
	bArm1HorzStn1SlantedLeft_12 AT %MX20004.12 : BOOL;
	bArm1HorzStn1SlantedLeft_13 AT %MX20004.13 : BOOL;
	bArm1HorzStn1SlantedLeft_14 AT %MX20004.14 : BOOL;
	bArm1HorzStn1SlantedLeft_15 AT %MX20004.15 : BOOL;
	bArm1HorzStn1SlantedLeft_16 AT %MX20004.16 : BOOL;
	bArm1HorzStn1SlantedLeft_17 AT %MX20004.17 : BOOL;
	bArm1HorzStn1SlantedLeft_18 AT %MX20004.18 : BOOL;
	bArm1HorzStn1SlantedLeft_19 AT %MX20004.19 : BOOL;
	bArm1HorzStn1SlantedLeft_20 AT %MX20004.20 : BOOL;
	bArm1HorzStn1SlantedLeft_21 AT %MX20004.21 : BOOL;
	bArm1HorzStn1SlantedLeft_22 AT %MX20004.22 : BOOL;
	bArm1HorzStn1SlantedLeft_23 AT %MX20004.23 : BOOL;
	bArm1HorzStn1SlantedLeft_24 AT %MX20004.24 : BOOL;
	bArm1HorzStn1SlantedLeft_25 AT %MX20004.25 : BOOL;
	bArm1HorzStn1SlantedLeft_26 AT %MX20004.26 : BOOL;
	bArm1HorzStn1SlantedLeft_27 AT %MX20004.27 : BOOL;
	bArm1HorzStn1SlantedLeft_28 AT %MX20004.28 : BOOL;
	bArm1HorzStn1SlantedLeft_29 AT %MX20004.29 : BOOL;
	bArm1HorzStn1SlantedLeft_30 AT %MX20004.30 : BOOL;
	bArm1HorzStn1SlantedLeft_31 AT %MX20004.31 : BOOL;

	bArm1HorzStn2SlantedLeft_00 AT %MX20008.0 : BOOL;
	bArm1HorzStn2SlantedLeft_01 AT %MX20008.1 : BOOL;
	bArm1HorzStn2SlantedLeft_02 AT %MX20008.2 : BOOL;
	bArm1HorzStn2SlantedLeft_03 AT %MX20008.3 : BOOL;
	bArm1HorzStn2SlantedLeft_04 AT %MX20008.4 : BOOL;
	bArm1HorzStn2SlantedLeft_05 AT %MX20008.5 : BOOL;
	bArm1HorzStn2SlantedLeft_06 AT %MX20008.6 : BOOL;
	bArm1HorzStn2SlantedLeft_07 AT %MX20008.7 : BOOL;
	bArm1HorzStn2SlantedLeft_08 AT %MX20008.8 : BOOL;
	bArm1HorzStn2SlantedLeft_09 AT %MX20008.9 : BOOL;
	bArm1HorzStn2SlantedLeft_10 AT %MX20008.10 : BOOL;
	bArm1HorzStn2SlantedLeft_11 AT %MX20008.11 : BOOL;
	bArm1HorzStn2SlantedLeft_12 AT %MX20008.12 : BOOL;
	bArm1HorzStn2SlantedLeft_13 AT %MX20008.13 : BOOL;
	bArm1HorzStn2SlantedLeft_14 AT %MX20008.14 : BOOL;
	bArm1HorzStn2SlantedLeft_15 AT %MX20008.15 : BOOL;
	bArm1HorzStn2SlantedLeft_16 AT %MX20008.16 : BOOL;
	bArm1HorzStn2SlantedLeft_17 AT %MX20008.17 : BOOL;
	bArm1HorzStn2SlantedLeft_18 AT %MX20008.18 : BOOL;
	bArm1HorzStn2SlantedLeft_19 AT %MX20008.19 : BOOL;
	bArm1HorzStn2SlantedLeft_20 AT %MX20008.20 : BOOL;
	bArm1HorzStn2SlantedLeft_21 AT %MX20008.21 : BOOL;
	bArm1HorzStn2SlantedLeft_22 AT %MX20008.22 : BOOL;
	bArm1HorzStn2SlantedLeft_23 AT %MX20008.23 : BOOL;
	bArm1HorzStn2SlantedLeft_24 AT %MX20008.24 : BOOL;
	bArm1HorzStn2SlantedLeft_25 AT %MX20008.25 : BOOL;
	bArm1HorzStn2SlantedLeft_26 AT %MX20008.26 : BOOL;
	bArm1HorzStn2SlantedLeft_27 AT %MX20008.27 : BOOL;
	bArm1HorzStn2SlantedLeft_28 AT %MX20008.28 : BOOL;
	bArm1HorzStn2SlantedLeft_29 AT %MX20008.29 : BOOL;
	bArm1HorzStn2SlantedLeft_30 AT %MX20008.30 : BOOL;
	bArm1HorzStn2SlantedLeft_31 AT %MX20008.31 : BOOL;

	bArm1HorzStn3SlantedLeft_00 AT %MX20012.0 : BOOL;
	bArm1HorzStn3SlantedLeft_01 AT %MX20012.1 : BOOL;
	bArm1HorzStn3SlantedLeft_02 AT %MX20012.2 : BOOL;
	bArm1HorzStn3SlantedLeft_03 AT %MX20012.3 : BOOL;
	bArm1HorzStn3SlantedLeft_04 AT %MX20012.4 : BOOL;
	bArm1HorzStn3SlantedLeft_05 AT %MX20012.5 : BOOL;
	bArm1HorzStn3SlantedLeft_06 AT %MX20012.6 : BOOL;
	bArm1HorzStn3SlantedLeft_07 AT %MX20012.7 : BOOL;
	bArm1HorzStn3SlantedLeft_08 AT %MX20012.8 : BOOL;
	bArm1HorzStn3SlantedLeft_09 AT %MX20012.9 : BOOL;
	bArm1HorzStn3SlantedLeft_10 AT %MX20012.10 : BOOL;
	bArm1HorzStn3SlantedLeft_11 AT %MX20012.11 : BOOL;
	bArm1HorzStn3SlantedLeft_12 AT %MX20012.12 : BOOL;
	bArm1HorzStn3SlantedLeft_13 AT %MX20012.13 : BOOL;
	bArm1HorzStn3SlantedLeft_14 AT %MX20012.14 : BOOL;
	bArm1HorzStn3SlantedLeft_15 AT %MX20012.15 : BOOL;
	bArm1HorzStn3SlantedLeft_16 AT %MX20012.16 : BOOL;
	bArm1HorzStn3SlantedLeft_17 AT %MX20012.17 : BOOL;
	bArm1HorzStn3SlantedLeft_18 AT %MX20012.18 : BOOL;
	bArm1HorzStn3SlantedLeft_19 AT %MX20012.19 : BOOL;
	bArm1HorzStn3SlantedLeft_20 AT %MX20012.20 : BOOL;
	bArm1HorzStn3SlantedLeft_21 AT %MX20012.21 : BOOL;
	bArm1HorzStn3SlantedLeft_22 AT %MX20012.22 : BOOL;
	bArm1HorzStn3SlantedLeft_23 AT %MX20012.23 : BOOL;
	bArm1HorzStn3SlantedLeft_24 AT %MX20012.24 : BOOL;
	bArm1HorzStn3SlantedLeft_25 AT %MX20012.25 : BOOL;
	bArm1HorzStn3SlantedLeft_26 AT %MX20012.26 : BOOL;
	bArm1HorzStn3SlantedLeft_27 AT %MX20012.27 : BOOL;
	bArm1HorzStn3SlantedLeft_28 AT %MX20012.28 : BOOL;
	bArm1HorzStn3SlantedLeft_29 AT %MX20012.29 : BOOL;
	bArm1HorzStn3SlantedLeft_30 AT %MX20012.30 : BOOL;
	bArm1HorzStn3SlantedLeft_31 AT %MX20012.31 : BOOL;

	bArm1HorzStn4SlantedLeft_00 AT %MX20016.0 : BOOL;
	bArm1HorzStn4SlantedLeft_01 AT %MX20016.1 : BOOL;
	bArm1HorzStn4SlantedLeft_02 AT %MX20016.2 : BOOL;
	bArm1HorzStn4SlantedLeft_03 AT %MX20016.3 : BOOL;
	bArm1HorzStn4SlantedLeft_04 AT %MX20016.4 : BOOL;
	bArm1HorzStn4SlantedLeft_05 AT %MX20016.5 : BOOL;
	bArm1HorzStn4SlantedLeft_06 AT %MX20016.6 : BOOL;
	bArm1HorzStn4SlantedLeft_07 AT %MX20016.7 : BOOL;
	bArm1HorzStn4SlantedLeft_08 AT %MX20016.8 : BOOL;
	bArm1HorzStn4SlantedLeft_09 AT %MX20016.9 : BOOL;
	bArm1HorzStn4SlantedLeft_10 AT %MX20016.10 : BOOL;
	bArm1HorzStn4SlantedLeft_11 AT %MX20016.11 : BOOL;
	bArm1HorzStn4SlantedLeft_12 AT %MX20016.12 : BOOL;
	bArm1HorzStn4SlantedLeft_13 AT %MX20016.13 : BOOL;
	bArm1HorzStn4SlantedLeft_14 AT %MX20016.14 : BOOL;
	bArm1HorzStn4SlantedLeft_15 AT %MX20016.15 : BOOL;
	bArm1HorzStn4SlantedLeft_16 AT %MX20016.16 : BOOL;
	bArm1HorzStn4SlantedLeft_17 AT %MX20016.17 : BOOL;
	bArm1HorzStn4SlantedLeft_18 AT %MX20016.18 : BOOL;
	bArm1HorzStn4SlantedLeft_19 AT %MX20016.19 : BOOL;
	bArm1HorzStn4SlantedLeft_20 AT %MX20016.20 : BOOL;
	bArm1HorzStn4SlantedLeft_21 AT %MX20016.21 : BOOL;
	bArm1HorzStn4SlantedLeft_22 AT %MX20016.22 : BOOL;
	bArm1HorzStn4SlantedLeft_23 AT %MX20016.23 : BOOL;
	bArm1HorzStn4SlantedLeft_24 AT %MX20016.24 : BOOL;
	bArm1HorzStn4SlantedLeft_25 AT %MX20016.25 : BOOL;
	bArm1HorzStn4SlantedLeft_26 AT %MX20016.26 : BOOL;
	bArm1HorzStn4SlantedLeft_27 AT %MX20016.27 : BOOL;
	bArm1HorzStn4SlantedLeft_28 AT %MX20016.28 : BOOL;
	bArm1HorzStn4SlantedLeft_29 AT %MX20016.29 : BOOL;
	bArm1HorzStn4SlantedLeft_30 AT %MX20016.30 : BOOL;
	bArm1HorzStn4SlantedLeft_31 AT %MX20016.31 : BOOL;

	bArm1HorzStn5SlantedLeft_00 AT %MX20020.0 : BOOL;
	bArm1HorzStn5SlantedLeft_01 AT %MX20020.1 : BOOL;
	bArm1HorzStn5SlantedLeft_02 AT %MX20020.2 : BOOL;
	bArm1HorzStn5SlantedLeft_03 AT %MX20020.3 : BOOL;
	bArm1HorzStn5SlantedLeft_04 AT %MX20020.4 : BOOL;
	bArm1HorzStn5SlantedLeft_05 AT %MX20020.5 : BOOL;
	bArm1HorzStn5SlantedLeft_06 AT %MX20020.6 : BOOL;
	bArm1HorzStn5SlantedLeft_07 AT %MX20020.7 : BOOL;
	bArm1HorzStn5SlantedLeft_08 AT %MX20020.8 : BOOL;
	bArm1HorzStn5SlantedLeft_09 AT %MX20020.9 : BOOL;
	bArm1HorzStn5SlantedLeft_10 AT %MX20020.10 : BOOL;
	bArm1HorzStn5SlantedLeft_11 AT %MX20020.11 : BOOL;
	bArm1HorzStn5SlantedLeft_12 AT %MX20020.12 : BOOL;
	bArm1HorzStn5SlantedLeft_13 AT %MX20020.13 : BOOL;
	bArm1HorzStn5SlantedLeft_14 AT %MX20020.14 : BOOL;
	bArm1HorzStn5SlantedLeft_15 AT %MX20020.15 : BOOL;
	bArm1HorzStn5SlantedLeft_16 AT %MX20020.16 : BOOL;
	bArm1HorzStn5SlantedLeft_17 AT %MX20020.17 : BOOL;
	bArm1HorzStn5SlantedLeft_18 AT %MX20020.18 : BOOL;
	bArm1HorzStn5SlantedLeft_19 AT %MX20020.19 : BOOL;
	bArm1HorzStn5SlantedLeft_20 AT %MX20020.20 : BOOL;
	bArm1HorzStn5SlantedLeft_21 AT %MX20020.21 : BOOL;
	bArm1HorzStn5SlantedLeft_22 AT %MX20020.22 : BOOL;
	bArm1HorzStn5SlantedLeft_23 AT %MX20020.23 : BOOL;
	bArm1HorzStn5SlantedLeft_24 AT %MX20020.24 : BOOL;
	bArm1HorzStn5SlantedLeft_25 AT %MX20020.25 : BOOL;
	bArm1HorzStn5SlantedLeft_26 AT %MX20020.26 : BOOL;
	bArm1HorzStn5SlantedLeft_27 AT %MX20020.27 : BOOL;
	bArm1HorzStn5SlantedLeft_28 AT %MX20020.28 : BOOL;
	bArm1HorzStn5SlantedLeft_29 AT %MX20020.29 : BOOL;
	bArm1HorzStn5SlantedLeft_30 AT %MX20020.30 : BOOL;
	bArm1HorzStn5SlantedLeft_31 AT %MX20020.31 : BOOL;

	bArm1HorzStn6SlantedLeft_00 AT %MX20024.0 : BOOL;
	bArm1HorzStn6SlantedLeft_01 AT %MX20024.1 : BOOL;
	bArm1HorzStn6SlantedLeft_02 AT %MX20024.2 : BOOL;
	bArm1HorzStn6SlantedLeft_03 AT %MX20024.3 : BOOL;
	bArm1HorzStn6SlantedLeft_04 AT %MX20024.4 : BOOL;
	bArm1HorzStn6SlantedLeft_05 AT %MX20024.5 : BOOL;
	bArm1HorzStn6SlantedLeft_06 AT %MX20024.6 : BOOL;
	bArm1HorzStn6SlantedLeft_07 AT %MX20024.7 : BOOL;
	bArm1HorzStn6SlantedLeft_08 AT %MX20024.8 : BOOL;
	bArm1HorzStn6SlantedLeft_09 AT %MX20024.9 : BOOL;
	bArm1HorzStn6SlantedLeft_10 AT %MX20024.10 : BOOL;
	bArm1HorzStn6SlantedLeft_11 AT %MX20024.11 : BOOL;
	bArm1HorzStn6SlantedLeft_12 AT %MX20024.12 : BOOL;
	bArm1HorzStn6SlantedLeft_13 AT %MX20024.13 : BOOL;
	bArm1HorzStn6SlantedLeft_14 AT %MX20024.14 : BOOL;
	bArm1HorzStn6SlantedLeft_15 AT %MX20024.15 : BOOL;
	bArm1HorzStn6SlantedLeft_16 AT %MX20024.16 : BOOL;
	bArm1HorzStn6SlantedLeft_17 AT %MX20024.17 : BOOL;
	bArm1HorzStn6SlantedLeft_18 AT %MX20024.18 : BOOL;
	bArm1HorzStn6SlantedLeft_19 AT %MX20024.19 : BOOL;
	bArm1HorzStn6SlantedLeft_20 AT %MX20024.20 : BOOL;
	bArm1HorzStn6SlantedLeft_21 AT %MX20024.21 : BOOL;
	bArm1HorzStn6SlantedLeft_22 AT %MX20024.22 : BOOL;
	bArm1HorzStn6SlantedLeft_23 AT %MX20024.23 : BOOL;
	bArm1HorzStn6SlantedLeft_24 AT %MX20024.24 : BOOL;
	bArm1HorzStn6SlantedLeft_25 AT %MX20024.25 : BOOL;
	bArm1HorzStn6SlantedLeft_26 AT %MX20024.26 : BOOL;
	bArm1HorzStn6SlantedLeft_27 AT %MX20024.27 : BOOL;
	bArm1HorzStn6SlantedLeft_28 AT %MX20024.28 : BOOL;
	bArm1HorzStn6SlantedLeft_29 AT %MX20024.29 : BOOL;
	bArm1HorzStn6SlantedLeft_30 AT %MX20024.30 : BOOL;
	bArm1HorzStn6SlantedLeft_31 AT %MX20024.31 : BOOL;

	bArm1HorzStn7SlantedLeft_00 AT %MX20028.0 : BOOL;
	bArm1HorzStn7SlantedLeft_01 AT %MX20028.1 : BOOL;
	bArm1HorzStn7SlantedLeft_02 AT %MX20028.2 : BOOL;
	bArm1HorzStn7SlantedLeft_03 AT %MX20028.3 : BOOL;
	bArm1HorzStn7SlantedLeft_04 AT %MX20028.4 : BOOL;
	bArm1HorzStn7SlantedLeft_05 AT %MX20028.5 : BOOL;
	bArm1HorzStn7SlantedLeft_06 AT %MX20028.6 : BOOL;
	bArm1HorzStn7SlantedLeft_07 AT %MX20028.7 : BOOL;
	bArm1HorzStn7SlantedLeft_08 AT %MX20028.8 : BOOL;
	bArm1HorzStn7SlantedLeft_09 AT %MX20028.9 : BOOL;
	bArm1HorzStn7SlantedLeft_10 AT %MX20028.10 : BOOL;
	bArm1HorzStn7SlantedLeft_11 AT %MX20028.11 : BOOL;
	bArm1HorzStn7SlantedLeft_12 AT %MX20028.12 : BOOL;
	bArm1HorzStn7SlantedLeft_13 AT %MX20028.13 : BOOL;
	bArm1HorzStn7SlantedLeft_14 AT %MX20028.14 : BOOL;
	bArm1HorzStn7SlantedLeft_15 AT %MX20028.15 : BOOL;
	bArm1HorzStn7SlantedLeft_16 AT %MX20028.16 : BOOL;
	bArm1HorzStn7SlantedLeft_17 AT %MX20028.17 : BOOL;
	bArm1HorzStn7SlantedLeft_18 AT %MX20028.18 : BOOL;
	bArm1HorzStn7SlantedLeft_19 AT %MX20028.19 : BOOL;
	bArm1HorzStn7SlantedLeft_20 AT %MX20028.20 : BOOL;
	bArm1HorzStn7SlantedLeft_21 AT %MX20028.21 : BOOL;
	bArm1HorzStn7SlantedLeft_22 AT %MX20028.22 : BOOL;
	bArm1HorzStn7SlantedLeft_23 AT %MX20028.23 : BOOL;
	bArm1HorzStn7SlantedLeft_24 AT %MX20028.24 : BOOL;
	bArm1HorzStn7SlantedLeft_25 AT %MX20028.25 : BOOL;
	bArm1HorzStn7SlantedLeft_26 AT %MX20028.26 : BOOL;
	bArm1HorzStn7SlantedLeft_27 AT %MX20028.27 : BOOL;
	bArm1HorzStn7SlantedLeft_28 AT %MX20028.28 : BOOL;
	bArm1HorzStn7SlantedLeft_29 AT %MX20028.29 : BOOL;
	bArm1HorzStn7SlantedLeft_30 AT %MX20028.30 : BOOL;
	bArm1HorzStn7SlantedLeft_31 AT %MX20028.31 : BOOL;

	bArm1HorzStn8SlantedLeft_00 AT %MX20032.0 : BOOL;
	bArm1HorzStn8SlantedLeft_01 AT %MX20032.1 : BOOL;
	bArm1HorzStn8SlantedLeft_02 AT %MX20032.2 : BOOL;
	bArm1HorzStn8SlantedLeft_03 AT %MX20032.3 : BOOL;
	bArm1HorzStn8SlantedLeft_04 AT %MX20032.4 : BOOL;
	bArm1HorzStn8SlantedLeft_05 AT %MX20032.5 : BOOL;
	bArm1HorzStn8SlantedLeft_06 AT %MX20032.6 : BOOL;
	bArm1HorzStn8SlantedLeft_07 AT %MX20032.7 : BOOL;
	bArm1HorzStn8SlantedLeft_08 AT %MX20032.8 : BOOL;
	bArm1HorzStn8SlantedLeft_09 AT %MX20032.9 : BOOL;
	bArm1HorzStn8SlantedLeft_10 AT %MX20032.10 : BOOL;
	bArm1HorzStn8SlantedLeft_11 AT %MX20032.11 : BOOL;
	bArm1HorzStn8SlantedLeft_12 AT %MX20032.12 : BOOL;
	bArm1HorzStn8SlantedLeft_13 AT %MX20032.13 : BOOL;
	bArm1HorzStn8SlantedLeft_14 AT %MX20032.14 : BOOL;
	bArm1HorzStn8SlantedLeft_15 AT %MX20032.15 : BOOL;
	bArm1HorzStn8SlantedLeft_16 AT %MX20032.16 : BOOL;
	bArm1HorzStn8SlantedLeft_17 AT %MX20032.17 : BOOL;
	bArm1HorzStn8SlantedLeft_18 AT %MX20032.18 : BOOL;
	bArm1HorzStn8SlantedLeft_19 AT %MX20032.19 : BOOL;
	bArm1HorzStn8SlantedLeft_20 AT %MX20032.20 : BOOL;
	bArm1HorzStn8SlantedLeft_21 AT %MX20032.21 : BOOL;
	bArm1HorzStn8SlantedLeft_22 AT %MX20032.22 : BOOL;
	bArm1HorzStn8SlantedLeft_23 AT %MX20032.23 : BOOL;
	bArm1HorzStn8SlantedLeft_24 AT %MX20032.24 : BOOL;
	bArm1HorzStn8SlantedLeft_25 AT %MX20032.25 : BOOL;
	bArm1HorzStn8SlantedLeft_26 AT %MX20032.26 : BOOL;
	bArm1HorzStn8SlantedLeft_27 AT %MX20032.27 : BOOL;
	bArm1HorzStn8SlantedLeft_28 AT %MX20032.28 : BOOL;
	bArm1HorzStn8SlantedLeft_29 AT %MX20032.29 : BOOL;
	bArm1HorzStn8SlantedLeft_30 AT %MX20032.30 : BOOL;
	bArm1HorzStn8SlantedLeft_31 AT %MX20032.31 : BOOL;

	bArm1HorzStn9SlantedLeft_00 AT %MX20036.0 : BOOL;
	bArm1HorzStn9SlantedLeft_01 AT %MX20036.1 : BOOL;
	bArm1HorzStn9SlantedLeft_02 AT %MX20036.2 : BOOL;
	bArm1HorzStn9SlantedLeft_03 AT %MX20036.3 : BOOL;
	bArm1HorzStn9SlantedLeft_04 AT %MX20036.4 : BOOL;
	bArm1HorzStn9SlantedLeft_05 AT %MX20036.5 : BOOL;
	bArm1HorzStn9SlantedLeft_06 AT %MX20036.6 : BOOL;
	bArm1HorzStn9SlantedLeft_07 AT %MX20036.7 : BOOL;
	bArm1HorzStn9SlantedLeft_08 AT %MX20036.8 : BOOL;
	bArm1HorzStn9SlantedLeft_09 AT %MX20036.9 : BOOL;
	bArm1HorzStn9SlantedLeft_10 AT %MX20036.10 : BOOL;
	bArm1HorzStn9SlantedLeft_11 AT %MX20036.11 : BOOL;
	bArm1HorzStn9SlantedLeft_12 AT %MX20036.12 : BOOL;
	bArm1HorzStn9SlantedLeft_13 AT %MX20036.13 : BOOL;
	bArm1HorzStn9SlantedLeft_14 AT %MX20036.14 : BOOL;
	bArm1HorzStn9SlantedLeft_15 AT %MX20036.15 : BOOL;
	bArm1HorzStn9SlantedLeft_16 AT %MX20036.16 : BOOL;
	bArm1HorzStn9SlantedLeft_17 AT %MX20036.17 : BOOL;
	bArm1HorzStn9SlantedLeft_18 AT %MX20036.18 : BOOL;
	bArm1HorzStn9SlantedLeft_19 AT %MX20036.19 : BOOL;
	bArm1HorzStn9SlantedLeft_20 AT %MX20036.20 : BOOL;
	bArm1HorzStn9SlantedLeft_21 AT %MX20036.21 : BOOL;
	bArm1HorzStn9SlantedLeft_22 AT %MX20036.22 : BOOL;
	bArm1HorzStn9SlantedLeft_23 AT %MX20036.23 : BOOL;
	bArm1HorzStn9SlantedLeft_24 AT %MX20036.24 : BOOL;
	bArm1HorzStn9SlantedLeft_25 AT %MX20036.25 : BOOL;
	bArm1HorzStn9SlantedLeft_26 AT %MX20036.26 : BOOL;
	bArm1HorzStn9SlantedLeft_27 AT %MX20036.27 : BOOL;
	bArm1HorzStn9SlantedLeft_28 AT %MX20036.28 : BOOL;
	bArm1HorzStn9SlantedLeft_29 AT %MX20036.29 : BOOL;
	bArm1HorzStn9SlantedLeft_30 AT %MX20036.30 : BOOL;
	bArm1HorzStn9SlantedLeft_31 AT %MX20036.31 : BOOL;

	bArm1HorzStn10SlantedLeft_00 AT %MX20040.0 : BOOL;
	bArm1HorzStn10SlantedLeft_01 AT %MX20040.1 : BOOL;
	bArm1HorzStn10SlantedLeft_02 AT %MX20040.2 : BOOL;
	bArm1HorzStn10SlantedLeft_03 AT %MX20040.3 : BOOL;
	bArm1HorzStn10SlantedLeft_04 AT %MX20040.4 : BOOL;
	bArm1HorzStn10SlantedLeft_05 AT %MX20040.5 : BOOL;
	bArm1HorzStn10SlantedLeft_06 AT %MX20040.6 : BOOL;
	bArm1HorzStn10SlantedLeft_07 AT %MX20040.7 : BOOL;
	bArm1HorzStn10SlantedLeft_08 AT %MX20040.8 : BOOL;
	bArm1HorzStn10SlantedLeft_09 AT %MX20040.9 : BOOL;
	bArm1HorzStn10SlantedLeft_10 AT %MX20040.10 : BOOL;
	bArm1HorzStn10SlantedLeft_11 AT %MX20040.11 : BOOL;
	bArm1HorzStn10SlantedLeft_12 AT %MX20040.12 : BOOL;
	bArm1HorzStn10SlantedLeft_13 AT %MX20040.13 : BOOL;
	bArm1HorzStn10SlantedLeft_14 AT %MX20040.14 : BOOL;
	bArm1HorzStn10SlantedLeft_15 AT %MX20040.15 : BOOL;
	bArm1HorzStn10SlantedLeft_16 AT %MX20040.16 : BOOL;
	bArm1HorzStn10SlantedLeft_17 AT %MX20040.17 : BOOL;
	bArm1HorzStn10SlantedLeft_18 AT %MX20040.18 : BOOL;
	bArm1HorzStn10SlantedLeft_19 AT %MX20040.19 : BOOL;
	bArm1HorzStn10SlantedLeft_20 AT %MX20040.20 : BOOL;
	bArm1HorzStn10SlantedLeft_21 AT %MX20040.21 : BOOL;
	bArm1HorzStn10SlantedLeft_22 AT %MX20040.22 : BOOL;
	bArm1HorzStn10SlantedLeft_23 AT %MX20040.23 : BOOL;
	bArm1HorzStn10SlantedLeft_24 AT %MX20040.24 : BOOL;
	bArm1HorzStn10SlantedLeft_25 AT %MX20040.25 : BOOL;
	bArm1HorzStn10SlantedLeft_26 AT %MX20040.26 : BOOL;
	bArm1HorzStn10SlantedLeft_27 AT %MX20040.27 : BOOL;
	bArm1HorzStn10SlantedLeft_28 AT %MX20040.28 : BOOL;
	bArm1HorzStn10SlantedLeft_29 AT %MX20040.29 : BOOL;
	bArm1HorzStn10SlantedLeft_30 AT %MX20040.30 : BOOL;
	bArm1HorzStn10SlantedLeft_31 AT %MX20040.31 : BOOL;

	bArm1HorzStn11SlantedLeft_00 AT %MX20044.0 : BOOL;
	bArm1HorzStn11SlantedLeft_01 AT %MX20044.1 : BOOL;
	bArm1HorzStn11SlantedLeft_02 AT %MX20044.2 : BOOL;
	bArm1HorzStn11SlantedLeft_03 AT %MX20044.3 : BOOL;
	bArm1HorzStn11SlantedLeft_04 AT %MX20044.4 : BOOL;
	bArm1HorzStn11SlantedLeft_05 AT %MX20044.5 : BOOL;
	bArm1HorzStn11SlantedLeft_06 AT %MX20044.6 : BOOL;
	bArm1HorzStn11SlantedLeft_07 AT %MX20044.7 : BOOL;
	bArm1HorzStn11SlantedLeft_08 AT %MX20044.8 : BOOL;
	bArm1HorzStn11SlantedLeft_09 AT %MX20044.9 : BOOL;
	bArm1HorzStn11SlantedLeft_10 AT %MX20044.10 : BOOL;
	bArm1HorzStn11SlantedLeft_11 AT %MX20044.11 : BOOL;
	bArm1HorzStn11SlantedLeft_12 AT %MX20044.12 : BOOL;
	bArm1HorzStn11SlantedLeft_13 AT %MX20044.13 : BOOL;
	bArm1HorzStn11SlantedLeft_14 AT %MX20044.14 : BOOL;
	bArm1HorzStn11SlantedLeft_15 AT %MX20044.15 : BOOL;
	bArm1HorzStn11SlantedLeft_16 AT %MX20044.16 : BOOL;
	bArm1HorzStn11SlantedLeft_17 AT %MX20044.17 : BOOL;
	bArm1HorzStn11SlantedLeft_18 AT %MX20044.18 : BOOL;
	bArm1HorzStn11SlantedLeft_19 AT %MX20044.19 : BOOL;
	bArm1HorzStn11SlantedLeft_20 AT %MX20044.20 : BOOL;
	bArm1HorzStn11SlantedLeft_21 AT %MX20044.21 : BOOL;
	bArm1HorzStn11SlantedLeft_22 AT %MX20044.22 : BOOL;
	bArm1HorzStn11SlantedLeft_23 AT %MX20044.23 : BOOL;
	bArm1HorzStn11SlantedLeft_24 AT %MX20044.24 : BOOL;
	bArm1HorzStn11SlantedLeft_25 AT %MX20044.25 : BOOL;
	bArm1HorzStn11SlantedLeft_26 AT %MX20044.26 : BOOL;
	bArm1HorzStn11SlantedLeft_27 AT %MX20044.27 : BOOL;
	bArm1HorzStn11SlantedLeft_28 AT %MX20044.28 : BOOL;
	bArm1HorzStn11SlantedLeft_29 AT %MX20044.29 : BOOL;
	bArm1HorzStn11SlantedLeft_30 AT %MX20044.30 : BOOL;
	bArm1HorzStn11SlantedLeft_31 AT %MX20044.31 : BOOL;

	bArm1HorzStn12SlantedLeft_00 AT %MX20048.0 : BOOL;
	bArm1HorzStn12SlantedLeft_01 AT %MX20048.1 : BOOL;
	bArm1HorzStn12SlantedLeft_02 AT %MX20048.2 : BOOL;
	bArm1HorzStn12SlantedLeft_03 AT %MX20048.3 : BOOL;
	bArm1HorzStn12SlantedLeft_04 AT %MX20048.4 : BOOL;
	bArm1HorzStn12SlantedLeft_05 AT %MX20048.5 : BOOL;
	bArm1HorzStn12SlantedLeft_06 AT %MX20048.6 : BOOL;
	bArm1HorzStn12SlantedLeft_07 AT %MX20048.7 : BOOL;
	bArm1HorzStn12SlantedLeft_08 AT %MX20048.8 : BOOL;
	bArm1HorzStn12SlantedLeft_09 AT %MX20048.9 : BOOL;
	bArm1HorzStn12SlantedLeft_10 AT %MX20048.10 : BOOL;
	bArm1HorzStn12SlantedLeft_11 AT %MX20048.11 : BOOL;
	bArm1HorzStn12SlantedLeft_12 AT %MX20048.12 : BOOL;
	bArm1HorzStn12SlantedLeft_13 AT %MX20048.13 : BOOL;
	bArm1HorzStn12SlantedLeft_14 AT %MX20048.14 : BOOL;
	bArm1HorzStn12SlantedLeft_15 AT %MX20048.15 : BOOL;
	bArm1HorzStn12SlantedLeft_16 AT %MX20048.16 : BOOL;
	bArm1HorzStn12SlantedLeft_17 AT %MX20048.17 : BOOL;
	bArm1HorzStn12SlantedLeft_18 AT %MX20048.18 : BOOL;
	bArm1HorzStn12SlantedLeft_19 AT %MX20048.19 : BOOL;
	bArm1HorzStn12SlantedLeft_20 AT %MX20048.20 : BOOL;
	bArm1HorzStn12SlantedLeft_21 AT %MX20048.21 : BOOL;
	bArm1HorzStn12SlantedLeft_22 AT %MX20048.22 : BOOL;
	bArm1HorzStn12SlantedLeft_23 AT %MX20048.23 : BOOL;
	bArm1HorzStn12SlantedLeft_24 AT %MX20048.24 : BOOL;
	bArm1HorzStn12SlantedLeft_25 AT %MX20048.25 : BOOL;
	bArm1HorzStn12SlantedLeft_26 AT %MX20048.26 : BOOL;
	bArm1HorzStn12SlantedLeft_27 AT %MX20048.27 : BOOL;
	bArm1HorzStn12SlantedLeft_28 AT %MX20048.28 : BOOL;
	bArm1HorzStn12SlantedLeft_29 AT %MX20048.29 : BOOL;
	bArm1HorzStn12SlantedLeft_30 AT %MX20048.30 : BOOL;
	bArm1HorzStn12SlantedLeft_31 AT %MX20048.31 : BOOL;


(*=============================== SlantedRight word ===============================*)
(*====================== SlantedRight BOOL LINK with %MX20100-MX20199 ======================*)

	bArm1HorzStn1SlantedRight_00 AT %MX20104.0 : BOOL;
	bArm1HorzStn1SlantedRight_01 AT %MX20104.1 : BOOL;
	bArm1HorzStn1SlantedRight_02 AT %MX20104.2 : BOOL;
	bArm1HorzStn1SlantedRight_03 AT %MX20104.3 : BOOL;
	bArm1HorzStn1SlantedRight_04 AT %MX20104.4 : BOOL;
	bArm1HorzStn1SlantedRight_05 AT %MX20104.5 : BOOL;
	bArm1HorzStn1SlantedRight_06 AT %MX20104.6 : BOOL;
	bArm1HorzStn1SlantedRight_07 AT %MX20104.7 : BOOL;
	bArm1HorzStn1SlantedRight_08 AT %MX20104.8 : BOOL;
	bArm1HorzStn1SlantedRight_09 AT %MX20104.9 : BOOL;
	bArm1HorzStn1SlantedRight_10 AT %MX20104.10 : BOOL;
	bArm1HorzStn1SlantedRight_11 AT %MX20104.11 : BOOL;
	bArm1HorzStn1SlantedRight_12 AT %MX20104.12 : BOOL;
	bArm1HorzStn1SlantedRight_13 AT %MX20104.13 : BOOL;
	bArm1HorzStn1SlantedRight_14 AT %MX20104.14 : BOOL;
	bArm1HorzStn1SlantedRight_15 AT %MX20104.15 : BOOL;
	bArm1HorzStn1SlantedRight_16 AT %MX20104.16 : BOOL;
	bArm1HorzStn1SlantedRight_17 AT %MX20104.17 : BOOL;
	bArm1HorzStn1SlantedRight_18 AT %MX20104.18 : BOOL;
	bArm1HorzStn1SlantedRight_19 AT %MX20104.19 : BOOL;
	bArm1HorzStn1SlantedRight_20 AT %MX20104.20 : BOOL;
	bArm1HorzStn1SlantedRight_21 AT %MX20104.21 : BOOL;
	bArm1HorzStn1SlantedRight_22 AT %MX20104.22 : BOOL;
	bArm1HorzStn1SlantedRight_23 AT %MX20104.23 : BOOL;
	bArm1HorzStn1SlantedRight_24 AT %MX20104.24 : BOOL;
	bArm1HorzStn1SlantedRight_25 AT %MX20104.25 : BOOL;
	bArm1HorzStn1SlantedRight_26 AT %MX20104.26 : BOOL;
	bArm1HorzStn1SlantedRight_27 AT %MX20104.27 : BOOL;
	bArm1HorzStn1SlantedRight_28 AT %MX20104.28 : BOOL;
	bArm1HorzStn1SlantedRight_29 AT %MX20104.29 : BOOL;
	bArm1HorzStn1SlantedRight_30 AT %MX20104.30 : BOOL;
	bArm1HorzStn1SlantedRight_31 AT %MX20104.31 : BOOL;

	bArm1HorzStn2SlantedRight_00 AT %MX20108.0 : BOOL;
	bArm1HorzStn2SlantedRight_01 AT %MX20108.1 : BOOL;
	bArm1HorzStn2SlantedRight_02 AT %MX20108.2 : BOOL;
	bArm1HorzStn2SlantedRight_03 AT %MX20108.3 : BOOL;
	bArm1HorzStn2SlantedRight_04 AT %MX20108.4 : BOOL;
	bArm1HorzStn2SlantedRight_05 AT %MX20108.5 : BOOL;
	bArm1HorzStn2SlantedRight_06 AT %MX20108.6 : BOOL;
	bArm1HorzStn2SlantedRight_07 AT %MX20108.7 : BOOL;
	bArm1HorzStn2SlantedRight_08 AT %MX20108.8 : BOOL;
	bArm1HorzStn2SlantedRight_09 AT %MX20108.9 : BOOL;
	bArm1HorzStn2SlantedRight_10 AT %MX20108.10 : BOOL;
	bArm1HorzStn2SlantedRight_11 AT %MX20108.11 : BOOL;
	bArm1HorzStn2SlantedRight_12 AT %MX20108.12 : BOOL;
	bArm1HorzStn2SlantedRight_13 AT %MX20108.13 : BOOL;
	bArm1HorzStn2SlantedRight_14 AT %MX20108.14 : BOOL;
	bArm1HorzStn2SlantedRight_15 AT %MX20108.15 : BOOL;
	bArm1HorzStn2SlantedRight_16 AT %MX20108.16 : BOOL;
	bArm1HorzStn2SlantedRight_17 AT %MX20108.17 : BOOL;
	bArm1HorzStn2SlantedRight_18 AT %MX20108.18 : BOOL;
	bArm1HorzStn2SlantedRight_19 AT %MX20108.19 : BOOL;
	bArm1HorzStn2SlantedRight_20 AT %MX20108.20 : BOOL;
	bArm1HorzStn2SlantedRight_21 AT %MX20108.21 : BOOL;
	bArm1HorzStn2SlantedRight_22 AT %MX20108.22 : BOOL;
	bArm1HorzStn2SlantedRight_23 AT %MX20108.23 : BOOL;
	bArm1HorzStn2SlantedRight_24 AT %MX20108.24 : BOOL;
	bArm1HorzStn2SlantedRight_25 AT %MX20108.25 : BOOL;
	bArm1HorzStn2SlantedRight_26 AT %MX20108.26 : BOOL;
	bArm1HorzStn2SlantedRight_27 AT %MX20108.27 : BOOL;
	bArm1HorzStn2SlantedRight_28 AT %MX20108.28 : BOOL;
	bArm1HorzStn2SlantedRight_29 AT %MX20108.29 : BOOL;
	bArm1HorzStn2SlantedRight_30 AT %MX20108.30 : BOOL;
	bArm1HorzStn2SlantedRight_31 AT %MX20108.31 : BOOL;

	bArm1HorzStn3SlantedRight_00 AT %MX20112.0 : BOOL;
	bArm1HorzStn3SlantedRight_01 AT %MX20112.1 : BOOL;
	bArm1HorzStn3SlantedRight_02 AT %MX20112.2 : BOOL;
	bArm1HorzStn3SlantedRight_03 AT %MX20112.3 : BOOL;
	bArm1HorzStn3SlantedRight_04 AT %MX20112.4 : BOOL;
	bArm1HorzStn3SlantedRight_05 AT %MX20112.5 : BOOL;
	bArm1HorzStn3SlantedRight_06 AT %MX20112.6 : BOOL;
	bArm1HorzStn3SlantedRight_07 AT %MX20112.7 : BOOL;
	bArm1HorzStn3SlantedRight_08 AT %MX20112.8 : BOOL;
	bArm1HorzStn3SlantedRight_09 AT %MX20112.9 : BOOL;
	bArm1HorzStn3SlantedRight_10 AT %MX20112.10 : BOOL;
	bArm1HorzStn3SlantedRight_11 AT %MX20112.11 : BOOL;
	bArm1HorzStn3SlantedRight_12 AT %MX20112.12 : BOOL;
	bArm1HorzStn3SlantedRight_13 AT %MX20112.13 : BOOL;
	bArm1HorzStn3SlantedRight_14 AT %MX20112.14 : BOOL;
	bArm1HorzStn3SlantedRight_15 AT %MX20112.15 : BOOL;
	bArm1HorzStn3SlantedRight_16 AT %MX20112.16 : BOOL;
	bArm1HorzStn3SlantedRight_17 AT %MX20112.17 : BOOL;
	bArm1HorzStn3SlantedRight_18 AT %MX20112.18 : BOOL;
	bArm1HorzStn3SlantedRight_19 AT %MX20112.19 : BOOL;
	bArm1HorzStn3SlantedRight_20 AT %MX20112.20 : BOOL;
	bArm1HorzStn3SlantedRight_21 AT %MX20112.21 : BOOL;
	bArm1HorzStn3SlantedRight_22 AT %MX20112.22 : BOOL;
	bArm1HorzStn3SlantedRight_23 AT %MX20112.23 : BOOL;
	bArm1HorzStn3SlantedRight_24 AT %MX20112.24 : BOOL;
	bArm1HorzStn3SlantedRight_25 AT %MX20112.25 : BOOL;
	bArm1HorzStn3SlantedRight_26 AT %MX20112.26 : BOOL;
	bArm1HorzStn3SlantedRight_27 AT %MX20112.27 : BOOL;
	bArm1HorzStn3SlantedRight_28 AT %MX20112.28 : BOOL;
	bArm1HorzStn3SlantedRight_29 AT %MX20112.29 : BOOL;
	bArm1HorzStn3SlantedRight_30 AT %MX20112.30 : BOOL;
	bArm1HorzStn3SlantedRight_31 AT %MX20112.31 : BOOL;

	bArm1HorzStn4SlantedRight_00 AT %MX20116.0 : BOOL;
	bArm1HorzStn4SlantedRight_01 AT %MX20116.1 : BOOL;
	bArm1HorzStn4SlantedRight_02 AT %MX20116.2 : BOOL;
	bArm1HorzStn4SlantedRight_03 AT %MX20116.3 : BOOL;
	bArm1HorzStn4SlantedRight_04 AT %MX20116.4 : BOOL;
	bArm1HorzStn4SlantedRight_05 AT %MX20116.5 : BOOL;
	bArm1HorzStn4SlantedRight_06 AT %MX20116.6 : BOOL;
	bArm1HorzStn4SlantedRight_07 AT %MX20116.7 : BOOL;
	bArm1HorzStn4SlantedRight_08 AT %MX20116.8 : BOOL;
	bArm1HorzStn4SlantedRight_09 AT %MX20116.9 : BOOL;
	bArm1HorzStn4SlantedRight_10 AT %MX20116.10 : BOOL;
	bArm1HorzStn4SlantedRight_11 AT %MX20116.11 : BOOL;
	bArm1HorzStn4SlantedRight_12 AT %MX20116.12 : BOOL;
	bArm1HorzStn4SlantedRight_13 AT %MX20116.13 : BOOL;
	bArm1HorzStn4SlantedRight_14 AT %MX20116.14 : BOOL;
	bArm1HorzStn4SlantedRight_15 AT %MX20116.15 : BOOL;
	bArm1HorzStn4SlantedRight_16 AT %MX20116.16 : BOOL;
	bArm1HorzStn4SlantedRight_17 AT %MX20116.17 : BOOL;
	bArm1HorzStn4SlantedRight_18 AT %MX20116.18 : BOOL;
	bArm1HorzStn4SlantedRight_19 AT %MX20116.19 : BOOL;
	bArm1HorzStn4SlantedRight_20 AT %MX20116.20 : BOOL;
	bArm1HorzStn4SlantedRight_21 AT %MX20116.21 : BOOL;
	bArm1HorzStn4SlantedRight_22 AT %MX20116.22 : BOOL;
	bArm1HorzStn4SlantedRight_23 AT %MX20116.23 : BOOL;
	bArm1HorzStn4SlantedRight_24 AT %MX20116.24 : BOOL;
	bArm1HorzStn4SlantedRight_25 AT %MX20116.25 : BOOL;
	bArm1HorzStn4SlantedRight_26 AT %MX20116.26 : BOOL;
	bArm1HorzStn4SlantedRight_27 AT %MX20116.27 : BOOL;
	bArm1HorzStn4SlantedRight_28 AT %MX20116.28 : BOOL;
	bArm1HorzStn4SlantedRight_29 AT %MX20116.29 : BOOL;
	bArm1HorzStn4SlantedRight_30 AT %MX20116.30 : BOOL;
	bArm1HorzStn4SlantedRight_31 AT %MX20116.31 : BOOL;

	bArm1HorzStn5SlantedRight_00 AT %MX20120.0 : BOOL;
	bArm1HorzStn5SlantedRight_01 AT %MX20120.1 : BOOL;
	bArm1HorzStn5SlantedRight_02 AT %MX20120.2 : BOOL;
	bArm1HorzStn5SlantedRight_03 AT %MX20120.3 : BOOL;
	bArm1HorzStn5SlantedRight_04 AT %MX20120.4 : BOOL;
	bArm1HorzStn5SlantedRight_05 AT %MX20120.5 : BOOL;
	bArm1HorzStn5SlantedRight_06 AT %MX20120.6 : BOOL;
	bArm1HorzStn5SlantedRight_07 AT %MX20120.7 : BOOL;
	bArm1HorzStn5SlantedRight_08 AT %MX20120.8 : BOOL;
	bArm1HorzStn5SlantedRight_09 AT %MX20120.9 : BOOL;
	bArm1HorzStn5SlantedRight_10 AT %MX20120.10 : BOOL;
	bArm1HorzStn5SlantedRight_11 AT %MX20120.11 : BOOL;
	bArm1HorzStn5SlantedRight_12 AT %MX20120.12 : BOOL;
	bArm1HorzStn5SlantedRight_13 AT %MX20120.13 : BOOL;
	bArm1HorzStn5SlantedRight_14 AT %MX20120.14 : BOOL;
	bArm1HorzStn5SlantedRight_15 AT %MX20120.15 : BOOL;
	bArm1HorzStn5SlantedRight_16 AT %MX20120.16 : BOOL;
	bArm1HorzStn5SlantedRight_17 AT %MX20120.17 : BOOL;
	bArm1HorzStn5SlantedRight_18 AT %MX20120.18 : BOOL;
	bArm1HorzStn5SlantedRight_19 AT %MX20120.19 : BOOL;
	bArm1HorzStn5SlantedRight_20 AT %MX20120.20 : BOOL;
	bArm1HorzStn5SlantedRight_21 AT %MX20120.21 : BOOL;
	bArm1HorzStn5SlantedRight_22 AT %MX20120.22 : BOOL;
	bArm1HorzStn5SlantedRight_23 AT %MX20120.23 : BOOL;
	bArm1HorzStn5SlantedRight_24 AT %MX20120.24 : BOOL;
	bArm1HorzStn5SlantedRight_25 AT %MX20120.25 : BOOL;
	bArm1HorzStn5SlantedRight_26 AT %MX20120.26 : BOOL;
	bArm1HorzStn5SlantedRight_27 AT %MX20120.27 : BOOL;
	bArm1HorzStn5SlantedRight_28 AT %MX20120.28 : BOOL;
	bArm1HorzStn5SlantedRight_29 AT %MX20120.29 : BOOL;
	bArm1HorzStn5SlantedRight_30 AT %MX20120.30 : BOOL;
	bArm1HorzStn5SlantedRight_31 AT %MX20120.31 : BOOL;

	bArm1HorzStn6SlantedRight_00 AT %MX20124.0 : BOOL;
	bArm1HorzStn6SlantedRight_01 AT %MX20124.1 : BOOL;
	bArm1HorzStn6SlantedRight_02 AT %MX20124.2 : BOOL;
	bArm1HorzStn6SlantedRight_03 AT %MX20124.3 : BOOL;
	bArm1HorzStn6SlantedRight_04 AT %MX20124.4 : BOOL;
	bArm1HorzStn6SlantedRight_05 AT %MX20124.5 : BOOL;
	bArm1HorzStn6SlantedRight_06 AT %MX20124.6 : BOOL;
	bArm1HorzStn6SlantedRight_07 AT %MX20124.7 : BOOL;
	bArm1HorzStn6SlantedRight_08 AT %MX20124.8 : BOOL;
	bArm1HorzStn6SlantedRight_09 AT %MX20124.9 : BOOL;
	bArm1HorzStn6SlantedRight_10 AT %MX20124.10 : BOOL;
	bArm1HorzStn6SlantedRight_11 AT %MX20124.11 : BOOL;
	bArm1HorzStn6SlantedRight_12 AT %MX20124.12 : BOOL;
	bArm1HorzStn6SlantedRight_13 AT %MX20124.13 : BOOL;
	bArm1HorzStn6SlantedRight_14 AT %MX20124.14 : BOOL;
	bArm1HorzStn6SlantedRight_15 AT %MX20124.15 : BOOL;
	bArm1HorzStn6SlantedRight_16 AT %MX20124.16 : BOOL;
	bArm1HorzStn6SlantedRight_17 AT %MX20124.17 : BOOL;
	bArm1HorzStn6SlantedRight_18 AT %MX20124.18 : BOOL;
	bArm1HorzStn6SlantedRight_19 AT %MX20124.19 : BOOL;
	bArm1HorzStn6SlantedRight_20 AT %MX20124.20 : BOOL;
	bArm1HorzStn6SlantedRight_21 AT %MX20124.21 : BOOL;
	bArm1HorzStn6SlantedRight_22 AT %MX20124.22 : BOOL;
	bArm1HorzStn6SlantedRight_23 AT %MX20124.23 : BOOL;
	bArm1HorzStn6SlantedRight_24 AT %MX20124.24 : BOOL;
	bArm1HorzStn6SlantedRight_25 AT %MX20124.25 : BOOL;
	bArm1HorzStn6SlantedRight_26 AT %MX20124.26 : BOOL;
	bArm1HorzStn6SlantedRight_27 AT %MX20124.27 : BOOL;
	bArm1HorzStn6SlantedRight_28 AT %MX20124.28 : BOOL;
	bArm1HorzStn6SlantedRight_29 AT %MX20124.29 : BOOL;
	bArm1HorzStn6SlantedRight_30 AT %MX20124.30 : BOOL;
	bArm1HorzStn6SlantedRight_31 AT %MX20124.31 : BOOL;

	bArm1HorzStn7SlantedRight_00 AT %MX20128.0 : BOOL;
	bArm1HorzStn7SlantedRight_01 AT %MX20128.1 : BOOL;
	bArm1HorzStn7SlantedRight_02 AT %MX20128.2 : BOOL;
	bArm1HorzStn7SlantedRight_03 AT %MX20128.3 : BOOL;
	bArm1HorzStn7SlantedRight_04 AT %MX20128.4 : BOOL;
	bArm1HorzStn7SlantedRight_05 AT %MX20128.5 : BOOL;
	bArm1HorzStn7SlantedRight_06 AT %MX20128.6 : BOOL;
	bArm1HorzStn7SlantedRight_07 AT %MX20128.7 : BOOL;
	bArm1HorzStn7SlantedRight_08 AT %MX20128.8 : BOOL;
	bArm1HorzStn7SlantedRight_09 AT %MX20128.9 : BOOL;
	bArm1HorzStn7SlantedRight_10 AT %MX20128.10 : BOOL;
	bArm1HorzStn7SlantedRight_11 AT %MX20128.11 : BOOL;
	bArm1HorzStn7SlantedRight_12 AT %MX20128.12 : BOOL;
	bArm1HorzStn7SlantedRight_13 AT %MX20128.13 : BOOL;
	bArm1HorzStn7SlantedRight_14 AT %MX20128.14 : BOOL;
	bArm1HorzStn7SlantedRight_15 AT %MX20128.15 : BOOL;
	bArm1HorzStn7SlantedRight_16 AT %MX20128.16 : BOOL;
	bArm1HorzStn7SlantedRight_17 AT %MX20128.17 : BOOL;
	bArm1HorzStn7SlantedRight_18 AT %MX20128.18 : BOOL;
	bArm1HorzStn7SlantedRight_19 AT %MX20128.19 : BOOL;
	bArm1HorzStn7SlantedRight_20 AT %MX20128.20 : BOOL;
	bArm1HorzStn7SlantedRight_21 AT %MX20128.21 : BOOL;
	bArm1HorzStn7SlantedRight_22 AT %MX20128.22 : BOOL;
	bArm1HorzStn7SlantedRight_23 AT %MX20128.23 : BOOL;
	bArm1HorzStn7SlantedRight_24 AT %MX20128.24 : BOOL;
	bArm1HorzStn7SlantedRight_25 AT %MX20128.25 : BOOL;
	bArm1HorzStn7SlantedRight_26 AT %MX20128.26 : BOOL;
	bArm1HorzStn7SlantedRight_27 AT %MX20128.27 : BOOL;
	bArm1HorzStn7SlantedRight_28 AT %MX20128.28 : BOOL;
	bArm1HorzStn7SlantedRight_29 AT %MX20128.29 : BOOL;
	bArm1HorzStn7SlantedRight_30 AT %MX20128.30 : BOOL;
	bArm1HorzStn7SlantedRight_31 AT %MX20128.31 : BOOL;

	bArm1HorzStn8SlantedRight_00 AT %MX20132.0 : BOOL;
	bArm1HorzStn8SlantedRight_01 AT %MX20132.1 : BOOL;
	bArm1HorzStn8SlantedRight_02 AT %MX20132.2 : BOOL;
	bArm1HorzStn8SlantedRight_03 AT %MX20132.3 : BOOL;
	bArm1HorzStn8SlantedRight_04 AT %MX20132.4 : BOOL;
	bArm1HorzStn8SlantedRight_05 AT %MX20132.5 : BOOL;
	bArm1HorzStn8SlantedRight_06 AT %MX20132.6 : BOOL;
	bArm1HorzStn8SlantedRight_07 AT %MX20132.7 : BOOL;
	bArm1HorzStn8SlantedRight_08 AT %MX20132.8 : BOOL;
	bArm1HorzStn8SlantedRight_09 AT %MX20132.9 : BOOL;
	bArm1HorzStn8SlantedRight_10 AT %MX20132.10 : BOOL;
	bArm1HorzStn8SlantedRight_11 AT %MX20132.11 : BOOL;
	bArm1HorzStn8SlantedRight_12 AT %MX20132.12 : BOOL;
	bArm1HorzStn8SlantedRight_13 AT %MX20132.13 : BOOL;
	bArm1HorzStn8SlantedRight_14 AT %MX20132.14 : BOOL;
	bArm1HorzStn8SlantedRight_15 AT %MX20132.15 : BOOL;
	bArm1HorzStn8SlantedRight_16 AT %MX20132.16 : BOOL;
	bArm1HorzStn8SlantedRight_17 AT %MX20132.17 : BOOL;
	bArm1HorzStn8SlantedRight_18 AT %MX20132.18 : BOOL;
	bArm1HorzStn8SlantedRight_19 AT %MX20132.19 : BOOL;
	bArm1HorzStn8SlantedRight_20 AT %MX20132.20 : BOOL;
	bArm1HorzStn8SlantedRight_21 AT %MX20132.21 : BOOL;
	bArm1HorzStn8SlantedRight_22 AT %MX20132.22 : BOOL;
	bArm1HorzStn8SlantedRight_23 AT %MX20132.23 : BOOL;
	bArm1HorzStn8SlantedRight_24 AT %MX20132.24 : BOOL;
	bArm1HorzStn8SlantedRight_25 AT %MX20132.25 : BOOL;
	bArm1HorzStn8SlantedRight_26 AT %MX20132.26 : BOOL;
	bArm1HorzStn8SlantedRight_27 AT %MX20132.27 : BOOL;
	bArm1HorzStn8SlantedRight_28 AT %MX20132.28 : BOOL;
	bArm1HorzStn8SlantedRight_29 AT %MX20132.29 : BOOL;
	bArm1HorzStn8SlantedRight_30 AT %MX20132.30 : BOOL;
	bArm1HorzStn8SlantedRight_31 AT %MX20132.31 : BOOL;

	bArm1HorzStn9SlantedRight_00 AT %MX20136.0 : BOOL;
	bArm1HorzStn9SlantedRight_01 AT %MX20136.1 : BOOL;
	bArm1HorzStn9SlantedRight_02 AT %MX20136.2 : BOOL;
	bArm1HorzStn9SlantedRight_03 AT %MX20136.3 : BOOL;
	bArm1HorzStn9SlantedRight_04 AT %MX20136.4 : BOOL;
	bArm1HorzStn9SlantedRight_05 AT %MX20136.5 : BOOL;
	bArm1HorzStn9SlantedRight_06 AT %MX20136.6 : BOOL;
	bArm1HorzStn9SlantedRight_07 AT %MX20136.7 : BOOL;
	bArm1HorzStn9SlantedRight_08 AT %MX20136.8 : BOOL;
	bArm1HorzStn9SlantedRight_09 AT %MX20136.9 : BOOL;
	bArm1HorzStn9SlantedRight_10 AT %MX20136.10 : BOOL;
	bArm1HorzStn9SlantedRight_11 AT %MX20136.11 : BOOL;
	bArm1HorzStn9SlantedRight_12 AT %MX20136.12 : BOOL;
	bArm1HorzStn9SlantedRight_13 AT %MX20136.13 : BOOL;
	bArm1HorzStn9SlantedRight_14 AT %MX20136.14 : BOOL;
	bArm1HorzStn9SlantedRight_15 AT %MX20136.15 : BOOL;
	bArm1HorzStn9SlantedRight_16 AT %MX20136.16 : BOOL;
	bArm1HorzStn9SlantedRight_17 AT %MX20136.17 : BOOL;
	bArm1HorzStn9SlantedRight_18 AT %MX20136.18 : BOOL;
	bArm1HorzStn9SlantedRight_19 AT %MX20136.19 : BOOL;
	bArm1HorzStn9SlantedRight_20 AT %MX20136.20 : BOOL;
	bArm1HorzStn9SlantedRight_21 AT %MX20136.21 : BOOL;
	bArm1HorzStn9SlantedRight_22 AT %MX20136.22 : BOOL;
	bArm1HorzStn9SlantedRight_23 AT %MX20136.23 : BOOL;
	bArm1HorzStn9SlantedRight_24 AT %MX20136.24 : BOOL;
	bArm1HorzStn9SlantedRight_25 AT %MX20136.25 : BOOL;
	bArm1HorzStn9SlantedRight_26 AT %MX20136.26 : BOOL;
	bArm1HorzStn9SlantedRight_27 AT %MX20136.27 : BOOL;
	bArm1HorzStn9SlantedRight_28 AT %MX20136.28 : BOOL;
	bArm1HorzStn9SlantedRight_29 AT %MX20136.29 : BOOL;
	bArm1HorzStn9SlantedRight_30 AT %MX20136.30 : BOOL;
	bArm1HorzStn9SlantedRight_31 AT %MX20136.31 : BOOL;

	bArm1HorzStn10SlantedRight_00 AT %MX20140.0 : BOOL;
	bArm1HorzStn10SlantedRight_01 AT %MX20140.1 : BOOL;
	bArm1HorzStn10SlantedRight_02 AT %MX20140.2 : BOOL;
	bArm1HorzStn10SlantedRight_03 AT %MX20140.3 : BOOL;
	bArm1HorzStn10SlantedRight_04 AT %MX20140.4 : BOOL;
	bArm1HorzStn10SlantedRight_05 AT %MX20140.5 : BOOL;
	bArm1HorzStn10SlantedRight_06 AT %MX20140.6 : BOOL;
	bArm1HorzStn10SlantedRight_07 AT %MX20140.7 : BOOL;
	bArm1HorzStn10SlantedRight_08 AT %MX20140.8 : BOOL;
	bArm1HorzStn10SlantedRight_09 AT %MX20140.9 : BOOL;
	bArm1HorzStn10SlantedRight_10 AT %MX20140.10 : BOOL;
	bArm1HorzStn10SlantedRight_11 AT %MX20140.11 : BOOL;
	bArm1HorzStn10SlantedRight_12 AT %MX20140.12 : BOOL;
	bArm1HorzStn10SlantedRight_13 AT %MX20140.13 : BOOL;
	bArm1HorzStn10SlantedRight_14 AT %MX20140.14 : BOOL;
	bArm1HorzStn10SlantedRight_15 AT %MX20140.15 : BOOL;
	bArm1HorzStn10SlantedRight_16 AT %MX20140.16 : BOOL;
	bArm1HorzStn10SlantedRight_17 AT %MX20140.17 : BOOL;
	bArm1HorzStn10SlantedRight_18 AT %MX20140.18 : BOOL;
	bArm1HorzStn10SlantedRight_19 AT %MX20140.19 : BOOL;
	bArm1HorzStn10SlantedRight_20 AT %MX20140.20 : BOOL;
	bArm1HorzStn10SlantedRight_21 AT %MX20140.21 : BOOL;
	bArm1HorzStn10SlantedRight_22 AT %MX20140.22 : BOOL;
	bArm1HorzStn10SlantedRight_23 AT %MX20140.23 : BOOL;
	bArm1HorzStn10SlantedRight_24 AT %MX20140.24 : BOOL;
	bArm1HorzStn10SlantedRight_25 AT %MX20140.25 : BOOL;
	bArm1HorzStn10SlantedRight_26 AT %MX20140.26 : BOOL;
	bArm1HorzStn10SlantedRight_27 AT %MX20140.27 : BOOL;
	bArm1HorzStn10SlantedRight_28 AT %MX20140.28 : BOOL;
	bArm1HorzStn10SlantedRight_29 AT %MX20140.29 : BOOL;
	bArm1HorzStn10SlantedRight_30 AT %MX20140.30 : BOOL;
	bArm1HorzStn10SlantedRight_31 AT %MX20140.31 : BOOL;

	bArm1HorzStn11SlantedRight_00 AT %MX20144.0 : BOOL;
	bArm1HorzStn11SlantedRight_01 AT %MX20144.1 : BOOL;
	bArm1HorzStn11SlantedRight_02 AT %MX20144.2 : BOOL;
	bArm1HorzStn11SlantedRight_03 AT %MX20144.3 : BOOL;
	bArm1HorzStn11SlantedRight_04 AT %MX20144.4 : BOOL;
	bArm1HorzStn11SlantedRight_05 AT %MX20144.5 : BOOL;
	bArm1HorzStn11SlantedRight_06 AT %MX20144.6 : BOOL;
	bArm1HorzStn11SlantedRight_07 AT %MX20144.7 : BOOL;
	bArm1HorzStn11SlantedRight_08 AT %MX20144.8 : BOOL;
	bArm1HorzStn11SlantedRight_09 AT %MX20144.9 : BOOL;
	bArm1HorzStn11SlantedRight_10 AT %MX20144.10 : BOOL;
	bArm1HorzStn11SlantedRight_11 AT %MX20144.11 : BOOL;
	bArm1HorzStn11SlantedRight_12 AT %MX20144.12 : BOOL;
	bArm1HorzStn11SlantedRight_13 AT %MX20144.13 : BOOL;
	bArm1HorzStn11SlantedRight_14 AT %MX20144.14 : BOOL;
	bArm1HorzStn11SlantedRight_15 AT %MX20144.15 : BOOL;
	bArm1HorzStn11SlantedRight_16 AT %MX20144.16 : BOOL;
	bArm1HorzStn11SlantedRight_17 AT %MX20144.17 : BOOL;
	bArm1HorzStn11SlantedRight_18 AT %MX20144.18 : BOOL;
	bArm1HorzStn11SlantedRight_19 AT %MX20144.19 : BOOL;
	bArm1HorzStn11SlantedRight_20 AT %MX20144.20 : BOOL;
	bArm1HorzStn11SlantedRight_21 AT %MX20144.21 : BOOL;
	bArm1HorzStn11SlantedRight_22 AT %MX20144.22 : BOOL;
	bArm1HorzStn11SlantedRight_23 AT %MX20144.23 : BOOL;
	bArm1HorzStn11SlantedRight_24 AT %MX20144.24 : BOOL;
	bArm1HorzStn11SlantedRight_25 AT %MX20144.25 : BOOL;
	bArm1HorzStn11SlantedRight_26 AT %MX20144.26 : BOOL;
	bArm1HorzStn11SlantedRight_27 AT %MX20144.27 : BOOL;
	bArm1HorzStn11SlantedRight_28 AT %MX20144.28 : BOOL;
	bArm1HorzStn11SlantedRight_29 AT %MX20144.29 : BOOL;
	bArm1HorzStn11SlantedRight_30 AT %MX20144.30 : BOOL;
	bArm1HorzStn11SlantedRight_31 AT %MX20144.31 : BOOL;

	bArm1HorzStn12SlantedRight_00 AT %MX20148.0 : BOOL;
	bArm1HorzStn12SlantedRight_01 AT %MX20148.1 : BOOL;
	bArm1HorzStn12SlantedRight_02 AT %MX20148.2 : BOOL;
	bArm1HorzStn12SlantedRight_03 AT %MX20148.3 : BOOL;
	bArm1HorzStn12SlantedRight_04 AT %MX20148.4 : BOOL;
	bArm1HorzStn12SlantedRight_05 AT %MX20148.5 : BOOL;
	bArm1HorzStn12SlantedRight_06 AT %MX20148.6 : BOOL;
	bArm1HorzStn12SlantedRight_07 AT %MX20148.7 : BOOL;
	bArm1HorzStn12SlantedRight_08 AT %MX20148.8 : BOOL;
	bArm1HorzStn12SlantedRight_09 AT %MX20148.9 : BOOL;
	bArm1HorzStn12SlantedRight_10 AT %MX20148.10 : BOOL;
	bArm1HorzStn12SlantedRight_11 AT %MX20148.11 : BOOL;
	bArm1HorzStn12SlantedRight_12 AT %MX20148.12 : BOOL;
	bArm1HorzStn12SlantedRight_13 AT %MX20148.13 : BOOL;
	bArm1HorzStn12SlantedRight_14 AT %MX20148.14 : BOOL;
	bArm1HorzStn12SlantedRight_15 AT %MX20148.15 : BOOL;
	bArm1HorzStn12SlantedRight_16 AT %MX20148.16 : BOOL;
	bArm1HorzStn12SlantedRight_17 AT %MX20148.17 : BOOL;
	bArm1HorzStn12SlantedRight_18 AT %MX20148.18 : BOOL;
	bArm1HorzStn12SlantedRight_19 AT %MX20148.19 : BOOL;
	bArm1HorzStn12SlantedRight_20 AT %MX20148.20 : BOOL;
	bArm1HorzStn12SlantedRight_21 AT %MX20148.21 : BOOL;
	bArm1HorzStn12SlantedRight_22 AT %MX20148.22 : BOOL;
	bArm1HorzStn12SlantedRight_23 AT %MX20148.23 : BOOL;
	bArm1HorzStn12SlantedRight_24 AT %MX20148.24 : BOOL;
	bArm1HorzStn12SlantedRight_25 AT %MX20148.25 : BOOL;
	bArm1HorzStn12SlantedRight_26 AT %MX20148.26 : BOOL;
	bArm1HorzStn12SlantedRight_27 AT %MX20148.27 : BOOL;
	bArm1HorzStn12SlantedRight_28 AT %MX20148.28 : BOOL;
	bArm1HorzStn12SlantedRight_29 AT %MX20148.29 : BOOL;
	bArm1HorzStn12SlantedRight_30 AT %MX20148.30 : BOOL;
	bArm1HorzStn12SlantedRight_31 AT %MX20148.31 : BOOL;


(*=============================== Hook word ===============================*)
(*====================== Hook BOOL LINK with %MX20200-MX20299 ======================*)

	bArm1HorzLD1Hook_00 AT %MX20252.0 : BOOL;
	bArm1HorzLD1Hook_01 AT %MX20252.1 : BOOL;
	bArm1HorzLD1Hook_02 AT %MX20252.2 : BOOL;
	bArm1HorzLD1Hook_03 AT %MX20252.3 : BOOL;
	bArm1HorzLD1Hook_04 AT %MX20252.4 : BOOL;
	bArm1HorzLD1Hook_05 AT %MX20252.5 : BOOL;
	bArm1HorzLD1Hook_06 AT %MX20252.6 : BOOL;
	bArm1HorzLD1Hook_07 AT %MX20252.7 : BOOL;
	bArm1HorzLD1Hook_08 AT %MX20252.8 : BOOL;
	bArm1HorzLD1Hook_09 AT %MX20252.9 : BOOL;
	bArm1HorzLD1Hook_10 AT %MX20252.10 : BOOL;
	bArm1HorzLD1Hook_11 AT %MX20252.11 : BOOL;
	bArm1HorzLD1Hook_12 AT %MX20252.12 : BOOL;
	bArm1HorzLD1Hook_13 AT %MX20252.13 : BOOL;
	bArm1HorzLD1Hook_14 AT %MX20252.14 : BOOL;
	bArm1HorzLD1Hook_15 AT %MX20252.15 : BOOL;
	bArm1HorzLD1Hook_16 AT %MX20252.16 : BOOL;
	bArm1HorzLD1Hook_17 AT %MX20252.17 : BOOL;
	bArm1HorzLD1Hook_18 AT %MX20252.18 : BOOL;
	bArm1HorzLD1Hook_19 AT %MX20252.19 : BOOL;
	bArm1HorzLD1Hook_20 AT %MX20252.20 : BOOL;
	bArm1HorzLD1Hook_21 AT %MX20252.21 : BOOL;
	bArm1HorzLD1Hook_22 AT %MX20252.22 : BOOL;
	bArm1HorzLD1Hook_23 AT %MX20252.23 : BOOL;
	bArm1HorzLD1Hook_24 AT %MX20252.24 : BOOL;
	bArm1HorzLD1Hook_25 AT %MX20252.25 : BOOL;
	bArm1HorzLD1Hook_26 AT %MX20252.26 : BOOL;
	bArm1HorzLD1Hook_27 AT %MX20252.27 : BOOL;
	bArm1HorzLD1Hook_28 AT %MX20252.28 : BOOL;
	bArm1HorzLD1Hook_29 AT %MX20252.29 : BOOL;
	bArm1HorzLD1Hook_30 AT %MX20252.30 : BOOL;
	bArm1HorzLD1Hook_31 AT %MX20252.31 : BOOL;

	bArm1HorzULD1Hook_00 AT %MX20256.0 : BOOL;
	bArm1HorzULD1Hook_01 AT %MX20256.1 : BOOL;
	bArm1HorzULD1Hook_02 AT %MX20256.2 : BOOL;
	bArm1HorzULD1Hook_03 AT %MX20256.3 : BOOL;
	bArm1HorzULD1Hook_04 AT %MX20256.4 : BOOL;
	bArm1HorzULD1Hook_05 AT %MX20256.5 : BOOL;
	bArm1HorzULD1Hook_06 AT %MX20256.6 : BOOL;
	bArm1HorzULD1Hook_07 AT %MX20256.7 : BOOL;
	bArm1HorzULD1Hook_08 AT %MX20256.8 : BOOL;
	bArm1HorzULD1Hook_09 AT %MX20256.9 : BOOL;
	bArm1HorzULD1Hook_10 AT %MX20256.10 : BOOL;
	bArm1HorzULD1Hook_11 AT %MX20256.11 : BOOL;
	bArm1HorzULD1Hook_12 AT %MX20256.12 : BOOL;
	bArm1HorzULD1Hook_13 AT %MX20256.13 : BOOL;
	bArm1HorzULD1Hook_14 AT %MX20256.14 : BOOL;
	bArm1HorzULD1Hook_15 AT %MX20256.15 : BOOL;
	bArm1HorzULD1Hook_16 AT %MX20256.16 : BOOL;
	bArm1HorzULD1Hook_17 AT %MX20256.17 : BOOL;
	bArm1HorzULD1Hook_18 AT %MX20256.18 : BOOL;
	bArm1HorzULD1Hook_19 AT %MX20256.19 : BOOL;
	bArm1HorzULD1Hook_20 AT %MX20256.20 : BOOL;
	bArm1HorzULD1Hook_21 AT %MX20256.21 : BOOL;
	bArm1HorzULD1Hook_22 AT %MX20256.22 : BOOL;
	bArm1HorzULD1Hook_23 AT %MX20256.23 : BOOL;
	bArm1HorzULD1Hook_24 AT %MX20256.24 : BOOL;
	bArm1HorzULD1Hook_25 AT %MX20256.25 : BOOL;
	bArm1HorzULD1Hook_26 AT %MX20256.26 : BOOL;
	bArm1HorzULD1Hook_27 AT %MX20256.27 : BOOL;
	bArm1HorzULD1Hook_28 AT %MX20256.28 : BOOL;
	bArm1HorzULD1Hook_29 AT %MX20256.29 : BOOL;
	bArm1HorzULD1Hook_30 AT %MX20256.30 : BOOL;
	bArm1HorzULD1Hook_31 AT %MX20256.31 : BOOL;

	bArm1HorzStn1Hook_00 AT %MX20204.0 : BOOL;
	bArm1HorzStn1Hook_01 AT %MX20204.1 : BOOL;
	bArm1HorzStn1Hook_02 AT %MX20204.2 : BOOL;
	bArm1HorzStn1Hook_03 AT %MX20204.3 : BOOL;
	bArm1HorzStn1Hook_04 AT %MX20204.4 : BOOL;
	bArm1HorzStn1Hook_05 AT %MX20204.5 : BOOL;
	bArm1HorzStn1Hook_06 AT %MX20204.6 : BOOL;
	bArm1HorzStn1Hook_07 AT %MX20204.7 : BOOL;
	bArm1HorzStn1Hook_08 AT %MX20204.8 : BOOL;
	bArm1HorzStn1Hook_09 AT %MX20204.9 : BOOL;
	bArm1HorzStn1Hook_10 AT %MX20204.10 : BOOL;
	bArm1HorzStn1Hook_11 AT %MX20204.11 : BOOL;
	bArm1HorzStn1Hook_12 AT %MX20204.12 : BOOL;
	bArm1HorzStn1Hook_13 AT %MX20204.13 : BOOL;
	bArm1HorzStn1Hook_14 AT %MX20204.14 : BOOL;
	bArm1HorzStn1Hook_15 AT %MX20204.15 : BOOL;
	bArm1HorzStn1Hook_16 AT %MX20204.16 : BOOL;
	bArm1HorzStn1Hook_17 AT %MX20204.17 : BOOL;
	bArm1HorzStn1Hook_18 AT %MX20204.18 : BOOL;
	bArm1HorzStn1Hook_19 AT %MX20204.19 : BOOL;
	bArm1HorzStn1Hook_20 AT %MX20204.20 : BOOL;
	bArm1HorzStn1Hook_21 AT %MX20204.21 : BOOL;
	bArm1HorzStn1Hook_22 AT %MX20204.22 : BOOL;
	bArm1HorzStn1Hook_23 AT %MX20204.23 : BOOL;
	bArm1HorzStn1Hook_24 AT %MX20204.24 : BOOL;
	bArm1HorzStn1Hook_25 AT %MX20204.25 : BOOL;
	bArm1HorzStn1Hook_26 AT %MX20204.26 : BOOL;
	bArm1HorzStn1Hook_27 AT %MX20204.27 : BOOL;
	bArm1HorzStn1Hook_28 AT %MX20204.28 : BOOL;
	bArm1HorzStn1Hook_29 AT %MX20204.29 : BOOL;
	bArm1HorzStn1Hook_30 AT %MX20204.30 : BOOL;
	bArm1HorzStn1Hook_31 AT %MX20204.31 : BOOL;

	bArm1HorzStn2Hook_00 AT %MX20208.0 : BOOL;
	bArm1HorzStn2Hook_01 AT %MX20208.1 : BOOL;
	bArm1HorzStn2Hook_02 AT %MX20208.2 : BOOL;
	bArm1HorzStn2Hook_03 AT %MX20208.3 : BOOL;
	bArm1HorzStn2Hook_04 AT %MX20208.4 : BOOL;
	bArm1HorzStn2Hook_05 AT %MX20208.5 : BOOL;
	bArm1HorzStn2Hook_06 AT %MX20208.6 : BOOL;
	bArm1HorzStn2Hook_07 AT %MX20208.7 : BOOL;
	bArm1HorzStn2Hook_08 AT %MX20208.8 : BOOL;
	bArm1HorzStn2Hook_09 AT %MX20208.9 : BOOL;
	bArm1HorzStn2Hook_10 AT %MX20208.10 : BOOL;
	bArm1HorzStn2Hook_11 AT %MX20208.11 : BOOL;
	bArm1HorzStn2Hook_12 AT %MX20208.12 : BOOL;
	bArm1HorzStn2Hook_13 AT %MX20208.13 : BOOL;
	bArm1HorzStn2Hook_14 AT %MX20208.14 : BOOL;
	bArm1HorzStn2Hook_15 AT %MX20208.15 : BOOL;
	bArm1HorzStn2Hook_16 AT %MX20208.16 : BOOL;
	bArm1HorzStn2Hook_17 AT %MX20208.17 : BOOL;
	bArm1HorzStn2Hook_18 AT %MX20208.18 : BOOL;
	bArm1HorzStn2Hook_19 AT %MX20208.19 : BOOL;
	bArm1HorzStn2Hook_20 AT %MX20208.20 : BOOL;
	bArm1HorzStn2Hook_21 AT %MX20208.21 : BOOL;
	bArm1HorzStn2Hook_22 AT %MX20208.22 : BOOL;
	bArm1HorzStn2Hook_23 AT %MX20208.23 : BOOL;
	bArm1HorzStn2Hook_24 AT %MX20208.24 : BOOL;
	bArm1HorzStn2Hook_25 AT %MX20208.25 : BOOL;
	bArm1HorzStn2Hook_26 AT %MX20208.26 : BOOL;
	bArm1HorzStn2Hook_27 AT %MX20208.27 : BOOL;
	bArm1HorzStn2Hook_28 AT %MX20208.28 : BOOL;
	bArm1HorzStn2Hook_29 AT %MX20208.29 : BOOL;
	bArm1HorzStn2Hook_30 AT %MX20208.30 : BOOL;
	bArm1HorzStn2Hook_31 AT %MX20208.31 : BOOL;

	bArm1HorzStn3Hook_00 AT %MX20212.0 : BOOL;
	bArm1HorzStn3Hook_01 AT %MX20212.1 : BOOL;
	bArm1HorzStn3Hook_02 AT %MX20212.2 : BOOL;
	bArm1HorzStn3Hook_03 AT %MX20212.3 : BOOL;
	bArm1HorzStn3Hook_04 AT %MX20212.4 : BOOL;
	bArm1HorzStn3Hook_05 AT %MX20212.5 : BOOL;
	bArm1HorzStn3Hook_06 AT %MX20212.6 : BOOL;
	bArm1HorzStn3Hook_07 AT %MX20212.7 : BOOL;
	bArm1HorzStn3Hook_08 AT %MX20212.8 : BOOL;
	bArm1HorzStn3Hook_09 AT %MX20212.9 : BOOL;
	bArm1HorzStn3Hook_10 AT %MX20212.10 : BOOL;
	bArm1HorzStn3Hook_11 AT %MX20212.11 : BOOL;
	bArm1HorzStn3Hook_12 AT %MX20212.12 : BOOL;
	bArm1HorzStn3Hook_13 AT %MX20212.13 : BOOL;
	bArm1HorzStn3Hook_14 AT %MX20212.14 : BOOL;
	bArm1HorzStn3Hook_15 AT %MX20212.15 : BOOL;
	bArm1HorzStn3Hook_16 AT %MX20212.16 : BOOL;
	bArm1HorzStn3Hook_17 AT %MX20212.17 : BOOL;
	bArm1HorzStn3Hook_18 AT %MX20212.18 : BOOL;
	bArm1HorzStn3Hook_19 AT %MX20212.19 : BOOL;
	bArm1HorzStn3Hook_20 AT %MX20212.20 : BOOL;
	bArm1HorzStn3Hook_21 AT %MX20212.21 : BOOL;
	bArm1HorzStn3Hook_22 AT %MX20212.22 : BOOL;
	bArm1HorzStn3Hook_23 AT %MX20212.23 : BOOL;
	bArm1HorzStn3Hook_24 AT %MX20212.24 : BOOL;
	bArm1HorzStn3Hook_25 AT %MX20212.25 : BOOL;
	bArm1HorzStn3Hook_26 AT %MX20212.26 : BOOL;
	bArm1HorzStn3Hook_27 AT %MX20212.27 : BOOL;
	bArm1HorzStn3Hook_28 AT %MX20212.28 : BOOL;
	bArm1HorzStn3Hook_29 AT %MX20212.29 : BOOL;
	bArm1HorzStn3Hook_30 AT %MX20212.30 : BOOL;
	bArm1HorzStn3Hook_31 AT %MX20212.31 : BOOL;

	bArm1HorzStn4Hook_00 AT %MX20216.0 : BOOL;
	bArm1HorzStn4Hook_01 AT %MX20216.1 : BOOL;
	bArm1HorzStn4Hook_02 AT %MX20216.2 : BOOL;
	bArm1HorzStn4Hook_03 AT %MX20216.3 : BOOL;
	bArm1HorzStn4Hook_04 AT %MX20216.4 : BOOL;
	bArm1HorzStn4Hook_05 AT %MX20216.5 : BOOL;
	bArm1HorzStn4Hook_06 AT %MX20216.6 : BOOL;
	bArm1HorzStn4Hook_07 AT %MX20216.7 : BOOL;
	bArm1HorzStn4Hook_08 AT %MX20216.8 : BOOL;
	bArm1HorzStn4Hook_09 AT %MX20216.9 : BOOL;
	bArm1HorzStn4Hook_10 AT %MX20216.10 : BOOL;
	bArm1HorzStn4Hook_11 AT %MX20216.11 : BOOL;
	bArm1HorzStn4Hook_12 AT %MX20216.12 : BOOL;
	bArm1HorzStn4Hook_13 AT %MX20216.13 : BOOL;
	bArm1HorzStn4Hook_14 AT %MX20216.14 : BOOL;
	bArm1HorzStn4Hook_15 AT %MX20216.15 : BOOL;
	bArm1HorzStn4Hook_16 AT %MX20216.16 : BOOL;
	bArm1HorzStn4Hook_17 AT %MX20216.17 : BOOL;
	bArm1HorzStn4Hook_18 AT %MX20216.18 : BOOL;
	bArm1HorzStn4Hook_19 AT %MX20216.19 : BOOL;
	bArm1HorzStn4Hook_20 AT %MX20216.20 : BOOL;
	bArm1HorzStn4Hook_21 AT %MX20216.21 : BOOL;
	bArm1HorzStn4Hook_22 AT %MX20216.22 : BOOL;
	bArm1HorzStn4Hook_23 AT %MX20216.23 : BOOL;
	bArm1HorzStn4Hook_24 AT %MX20216.24 : BOOL;
	bArm1HorzStn4Hook_25 AT %MX20216.25 : BOOL;
	bArm1HorzStn4Hook_26 AT %MX20216.26 : BOOL;
	bArm1HorzStn4Hook_27 AT %MX20216.27 : BOOL;
	bArm1HorzStn4Hook_28 AT %MX20216.28 : BOOL;
	bArm1HorzStn4Hook_29 AT %MX20216.29 : BOOL;
	bArm1HorzStn4Hook_30 AT %MX20216.30 : BOOL;
	bArm1HorzStn4Hook_31 AT %MX20216.31 : BOOL;

	bArm1HorzStn5Hook_00 AT %MX20220.0 : BOOL;
	bArm1HorzStn5Hook_01 AT %MX20220.1 : BOOL;
	bArm1HorzStn5Hook_02 AT %MX20220.2 : BOOL;
	bArm1HorzStn5Hook_03 AT %MX20220.3 : BOOL;
	bArm1HorzStn5Hook_04 AT %MX20220.4 : BOOL;
	bArm1HorzStn5Hook_05 AT %MX20220.5 : BOOL;
	bArm1HorzStn5Hook_06 AT %MX20220.6 : BOOL;
	bArm1HorzStn5Hook_07 AT %MX20220.7 : BOOL;
	bArm1HorzStn5Hook_08 AT %MX20220.8 : BOOL;
	bArm1HorzStn5Hook_09 AT %MX20220.9 : BOOL;
	bArm1HorzStn5Hook_10 AT %MX20220.10 : BOOL;
	bArm1HorzStn5Hook_11 AT %MX20220.11 : BOOL;
	bArm1HorzStn5Hook_12 AT %MX20220.12 : BOOL;
	bArm1HorzStn5Hook_13 AT %MX20220.13 : BOOL;
	bArm1HorzStn5Hook_14 AT %MX20220.14 : BOOL;
	bArm1HorzStn5Hook_15 AT %MX20220.15 : BOOL;
	bArm1HorzStn5Hook_16 AT %MX20220.16 : BOOL;
	bArm1HorzStn5Hook_17 AT %MX20220.17 : BOOL;
	bArm1HorzStn5Hook_18 AT %MX20220.18 : BOOL;
	bArm1HorzStn5Hook_19 AT %MX20220.19 : BOOL;
	bArm1HorzStn5Hook_20 AT %MX20220.20 : BOOL;
	bArm1HorzStn5Hook_21 AT %MX20220.21 : BOOL;
	bArm1HorzStn5Hook_22 AT %MX20220.22 : BOOL;
	bArm1HorzStn5Hook_23 AT %MX20220.23 : BOOL;
	bArm1HorzStn5Hook_24 AT %MX20220.24 : BOOL;
	bArm1HorzStn5Hook_25 AT %MX20220.25 : BOOL;
	bArm1HorzStn5Hook_26 AT %MX20220.26 : BOOL;
	bArm1HorzStn5Hook_27 AT %MX20220.27 : BOOL;
	bArm1HorzStn5Hook_28 AT %MX20220.28 : BOOL;
	bArm1HorzStn5Hook_29 AT %MX20220.29 : BOOL;
	bArm1HorzStn5Hook_30 AT %MX20220.30 : BOOL;
	bArm1HorzStn5Hook_31 AT %MX20220.31 : BOOL;

	bArm1HorzStn6Hook_00 AT %MX20224.0 : BOOL;
	bArm1HorzStn6Hook_01 AT %MX20224.1 : BOOL;
	bArm1HorzStn6Hook_02 AT %MX20224.2 : BOOL;
	bArm1HorzStn6Hook_03 AT %MX20224.3 : BOOL;
	bArm1HorzStn6Hook_04 AT %MX20224.4 : BOOL;
	bArm1HorzStn6Hook_05 AT %MX20224.5 : BOOL;
	bArm1HorzStn6Hook_06 AT %MX20224.6 : BOOL;
	bArm1HorzStn6Hook_07 AT %MX20224.7 : BOOL;
	bArm1HorzStn6Hook_08 AT %MX20224.8 : BOOL;
	bArm1HorzStn6Hook_09 AT %MX20224.9 : BOOL;
	bArm1HorzStn6Hook_10 AT %MX20224.10 : BOOL;
	bArm1HorzStn6Hook_11 AT %MX20224.11 : BOOL;
	bArm1HorzStn6Hook_12 AT %MX20224.12 : BOOL;
	bArm1HorzStn6Hook_13 AT %MX20224.13 : BOOL;
	bArm1HorzStn6Hook_14 AT %MX20224.14 : BOOL;
	bArm1HorzStn6Hook_15 AT %MX20224.15 : BOOL;
	bArm1HorzStn6Hook_16 AT %MX20224.16 : BOOL;
	bArm1HorzStn6Hook_17 AT %MX20224.17 : BOOL;
	bArm1HorzStn6Hook_18 AT %MX20224.18 : BOOL;
	bArm1HorzStn6Hook_19 AT %MX20224.19 : BOOL;
	bArm1HorzStn6Hook_20 AT %MX20224.20 : BOOL;
	bArm1HorzStn6Hook_21 AT %MX20224.21 : BOOL;
	bArm1HorzStn6Hook_22 AT %MX20224.22 : BOOL;
	bArm1HorzStn6Hook_23 AT %MX20224.23 : BOOL;
	bArm1HorzStn6Hook_24 AT %MX20224.24 : BOOL;
	bArm1HorzStn6Hook_25 AT %MX20224.25 : BOOL;
	bArm1HorzStn6Hook_26 AT %MX20224.26 : BOOL;
	bArm1HorzStn6Hook_27 AT %MX20224.27 : BOOL;
	bArm1HorzStn6Hook_28 AT %MX20224.28 : BOOL;
	bArm1HorzStn6Hook_29 AT %MX20224.29 : BOOL;
	bArm1HorzStn6Hook_30 AT %MX20224.30 : BOOL;
	bArm1HorzStn6Hook_31 AT %MX20224.31 : BOOL;

	bArm1HorzStn7Hook_00 AT %MX20228.0 : BOOL;
	bArm1HorzStn7Hook_01 AT %MX20228.1 : BOOL;
	bArm1HorzStn7Hook_02 AT %MX20228.2 : BOOL;
	bArm1HorzStn7Hook_03 AT %MX20228.3 : BOOL;
	bArm1HorzStn7Hook_04 AT %MX20228.4 : BOOL;
	bArm1HorzStn7Hook_05 AT %MX20228.5 : BOOL;
	bArm1HorzStn7Hook_06 AT %MX20228.6 : BOOL;
	bArm1HorzStn7Hook_07 AT %MX20228.7 : BOOL;
	bArm1HorzStn7Hook_08 AT %MX20228.8 : BOOL;
	bArm1HorzStn7Hook_09 AT %MX20228.9 : BOOL;
	bArm1HorzStn7Hook_10 AT %MX20228.10 : BOOL;
	bArm1HorzStn7Hook_11 AT %MX20228.11 : BOOL;
	bArm1HorzStn7Hook_12 AT %MX20228.12 : BOOL;
	bArm1HorzStn7Hook_13 AT %MX20228.13 : BOOL;
	bArm1HorzStn7Hook_14 AT %MX20228.14 : BOOL;
	bArm1HorzStn7Hook_15 AT %MX20228.15 : BOOL;
	bArm1HorzStn7Hook_16 AT %MX20228.16 : BOOL;
	bArm1HorzStn7Hook_17 AT %MX20228.17 : BOOL;
	bArm1HorzStn7Hook_18 AT %MX20228.18 : BOOL;
	bArm1HorzStn7Hook_19 AT %MX20228.19 : BOOL;
	bArm1HorzStn7Hook_20 AT %MX20228.20 : BOOL;
	bArm1HorzStn7Hook_21 AT %MX20228.21 : BOOL;
	bArm1HorzStn7Hook_22 AT %MX20228.22 : BOOL;
	bArm1HorzStn7Hook_23 AT %MX20228.23 : BOOL;
	bArm1HorzStn7Hook_24 AT %MX20228.24 : BOOL;
	bArm1HorzStn7Hook_25 AT %MX20228.25 : BOOL;
	bArm1HorzStn7Hook_26 AT %MX20228.26 : BOOL;
	bArm1HorzStn7Hook_27 AT %MX20228.27 : BOOL;
	bArm1HorzStn7Hook_28 AT %MX20228.28 : BOOL;
	bArm1HorzStn7Hook_29 AT %MX20228.29 : BOOL;
	bArm1HorzStn7Hook_30 AT %MX20228.30 : BOOL;
	bArm1HorzStn7Hook_31 AT %MX20228.31 : BOOL;

	bArm1HorzStn8Hook_00 AT %MX20232.0 : BOOL;
	bArm1HorzStn8Hook_01 AT %MX20232.1 : BOOL;
	bArm1HorzStn8Hook_02 AT %MX20232.2 : BOOL;
	bArm1HorzStn8Hook_03 AT %MX20232.3 : BOOL;
	bArm1HorzStn8Hook_04 AT %MX20232.4 : BOOL;
	bArm1HorzStn8Hook_05 AT %MX20232.5 : BOOL;
	bArm1HorzStn8Hook_06 AT %MX20232.6 : BOOL;
	bArm1HorzStn8Hook_07 AT %MX20232.7 : BOOL;
	bArm1HorzStn8Hook_08 AT %MX20232.8 : BOOL;
	bArm1HorzStn8Hook_09 AT %MX20232.9 : BOOL;
	bArm1HorzStn8Hook_10 AT %MX20232.10 : BOOL;
	bArm1HorzStn8Hook_11 AT %MX20232.11 : BOOL;
	bArm1HorzStn8Hook_12 AT %MX20232.12 : BOOL;
	bArm1HorzStn8Hook_13 AT %MX20232.13 : BOOL;
	bArm1HorzStn8Hook_14 AT %MX20232.14 : BOOL;
	bArm1HorzStn8Hook_15 AT %MX20232.15 : BOOL;
	bArm1HorzStn8Hook_16 AT %MX20232.16 : BOOL;
	bArm1HorzStn8Hook_17 AT %MX20232.17 : BOOL;
	bArm1HorzStn8Hook_18 AT %MX20232.18 : BOOL;
	bArm1HorzStn8Hook_19 AT %MX20232.19 : BOOL;
	bArm1HorzStn8Hook_20 AT %MX20232.20 : BOOL;
	bArm1HorzStn8Hook_21 AT %MX20232.21 : BOOL;
	bArm1HorzStn8Hook_22 AT %MX20232.22 : BOOL;
	bArm1HorzStn8Hook_23 AT %MX20232.23 : BOOL;
	bArm1HorzStn8Hook_24 AT %MX20232.24 : BOOL;
	bArm1HorzStn8Hook_25 AT %MX20232.25 : BOOL;
	bArm1HorzStn8Hook_26 AT %MX20232.26 : BOOL;
	bArm1HorzStn8Hook_27 AT %MX20232.27 : BOOL;
	bArm1HorzStn8Hook_28 AT %MX20232.28 : BOOL;
	bArm1HorzStn8Hook_29 AT %MX20232.29 : BOOL;
	bArm1HorzStn8Hook_30 AT %MX20232.30 : BOOL;
	bArm1HorzStn8Hook_31 AT %MX20232.31 : BOOL;

	bArm1HorzStn9Hook_00 AT %MX20236.0 : BOOL;
	bArm1HorzStn9Hook_01 AT %MX20236.1 : BOOL;
	bArm1HorzStn9Hook_02 AT %MX20236.2 : BOOL;
	bArm1HorzStn9Hook_03 AT %MX20236.3 : BOOL;
	bArm1HorzStn9Hook_04 AT %MX20236.4 : BOOL;
	bArm1HorzStn9Hook_05 AT %MX20236.5 : BOOL;
	bArm1HorzStn9Hook_06 AT %MX20236.6 : BOOL;
	bArm1HorzStn9Hook_07 AT %MX20236.7 : BOOL;
	bArm1HorzStn9Hook_08 AT %MX20236.8 : BOOL;
	bArm1HorzStn9Hook_09 AT %MX20236.9 : BOOL;
	bArm1HorzStn9Hook_10 AT %MX20236.10 : BOOL;
	bArm1HorzStn9Hook_11 AT %MX20236.11 : BOOL;
	bArm1HorzStn9Hook_12 AT %MX20236.12 : BOOL;
	bArm1HorzStn9Hook_13 AT %MX20236.13 : BOOL;
	bArm1HorzStn9Hook_14 AT %MX20236.14 : BOOL;
	bArm1HorzStn9Hook_15 AT %MX20236.15 : BOOL;
	bArm1HorzStn9Hook_16 AT %MX20236.16 : BOOL;
	bArm1HorzStn9Hook_17 AT %MX20236.17 : BOOL;
	bArm1HorzStn9Hook_18 AT %MX20236.18 : BOOL;
	bArm1HorzStn9Hook_19 AT %MX20236.19 : BOOL;
	bArm1HorzStn9Hook_20 AT %MX20236.20 : BOOL;
	bArm1HorzStn9Hook_21 AT %MX20236.21 : BOOL;
	bArm1HorzStn9Hook_22 AT %MX20236.22 : BOOL;
	bArm1HorzStn9Hook_23 AT %MX20236.23 : BOOL;
	bArm1HorzStn9Hook_24 AT %MX20236.24 : BOOL;
	bArm1HorzStn9Hook_25 AT %MX20236.25 : BOOL;
	bArm1HorzStn9Hook_26 AT %MX20236.26 : BOOL;
	bArm1HorzStn9Hook_27 AT %MX20236.27 : BOOL;
	bArm1HorzStn9Hook_28 AT %MX20236.28 : BOOL;
	bArm1HorzStn9Hook_29 AT %MX20236.29 : BOOL;
	bArm1HorzStn9Hook_30 AT %MX20236.30 : BOOL;
	bArm1HorzStn9Hook_31 AT %MX20236.31 : BOOL;

	bArm1HorzStn10Hook_00 AT %MX20240.0 : BOOL;
	bArm1HorzStn10Hook_01 AT %MX20240.1 : BOOL;
	bArm1HorzStn10Hook_02 AT %MX20240.2 : BOOL;
	bArm1HorzStn10Hook_03 AT %MX20240.3 : BOOL;
	bArm1HorzStn10Hook_04 AT %MX20240.4 : BOOL;
	bArm1HorzStn10Hook_05 AT %MX20240.5 : BOOL;
	bArm1HorzStn10Hook_06 AT %MX20240.6 : BOOL;
	bArm1HorzStn10Hook_07 AT %MX20240.7 : BOOL;
	bArm1HorzStn10Hook_08 AT %MX20240.8 : BOOL;
	bArm1HorzStn10Hook_09 AT %MX20240.9 : BOOL;
	bArm1HorzStn10Hook_10 AT %MX20240.10 : BOOL;
	bArm1HorzStn10Hook_11 AT %MX20240.11 : BOOL;
	bArm1HorzStn10Hook_12 AT %MX20240.12 : BOOL;
	bArm1HorzStn10Hook_13 AT %MX20240.13 : BOOL;
	bArm1HorzStn10Hook_14 AT %MX20240.14 : BOOL;
	bArm1HorzStn10Hook_15 AT %MX20240.15 : BOOL;
	bArm1HorzStn10Hook_16 AT %MX20240.16 : BOOL;
	bArm1HorzStn10Hook_17 AT %MX20240.17 : BOOL;
	bArm1HorzStn10Hook_18 AT %MX20240.18 : BOOL;
	bArm1HorzStn10Hook_19 AT %MX20240.19 : BOOL;
	bArm1HorzStn10Hook_20 AT %MX20240.20 : BOOL;
	bArm1HorzStn10Hook_21 AT %MX20240.21 : BOOL;
	bArm1HorzStn10Hook_22 AT %MX20240.22 : BOOL;
	bArm1HorzStn10Hook_23 AT %MX20240.23 : BOOL;
	bArm1HorzStn10Hook_24 AT %MX20240.24 : BOOL;
	bArm1HorzStn10Hook_25 AT %MX20240.25 : BOOL;
	bArm1HorzStn10Hook_26 AT %MX20240.26 : BOOL;
	bArm1HorzStn10Hook_27 AT %MX20240.27 : BOOL;
	bArm1HorzStn10Hook_28 AT %MX20240.28 : BOOL;
	bArm1HorzStn10Hook_29 AT %MX20240.29 : BOOL;
	bArm1HorzStn10Hook_30 AT %MX20240.30 : BOOL;
	bArm1HorzStn10Hook_31 AT %MX20240.31 : BOOL;

	bArm1HorzStn11Hook_00 AT %MX20244.0 : BOOL;
	bArm1HorzStn11Hook_01 AT %MX20244.1 : BOOL;
	bArm1HorzStn11Hook_02 AT %MX20244.2 : BOOL;
	bArm1HorzStn11Hook_03 AT %MX20244.3 : BOOL;
	bArm1HorzStn11Hook_04 AT %MX20244.4 : BOOL;
	bArm1HorzStn11Hook_05 AT %MX20244.5 : BOOL;
	bArm1HorzStn11Hook_06 AT %MX20244.6 : BOOL;
	bArm1HorzStn11Hook_07 AT %MX20244.7 : BOOL;
	bArm1HorzStn11Hook_08 AT %MX20244.8 : BOOL;
	bArm1HorzStn11Hook_09 AT %MX20244.9 : BOOL;
	bArm1HorzStn11Hook_10 AT %MX20244.10 : BOOL;
	bArm1HorzStn11Hook_11 AT %MX20244.11 : BOOL;
	bArm1HorzStn11Hook_12 AT %MX20244.12 : BOOL;
	bArm1HorzStn11Hook_13 AT %MX20244.13 : BOOL;
	bArm1HorzStn11Hook_14 AT %MX20244.14 : BOOL;
	bArm1HorzStn11Hook_15 AT %MX20244.15 : BOOL;
	bArm1HorzStn11Hook_16 AT %MX20244.16 : BOOL;
	bArm1HorzStn11Hook_17 AT %MX20244.17 : BOOL;
	bArm1HorzStn11Hook_18 AT %MX20244.18 : BOOL;
	bArm1HorzStn11Hook_19 AT %MX20244.19 : BOOL;
	bArm1HorzStn11Hook_20 AT %MX20244.20 : BOOL;
	bArm1HorzStn11Hook_21 AT %MX20244.21 : BOOL;
	bArm1HorzStn11Hook_22 AT %MX20244.22 : BOOL;
	bArm1HorzStn11Hook_23 AT %MX20244.23 : BOOL;
	bArm1HorzStn11Hook_24 AT %MX20244.24 : BOOL;
	bArm1HorzStn11Hook_25 AT %MX20244.25 : BOOL;
	bArm1HorzStn11Hook_26 AT %MX20244.26 : BOOL;
	bArm1HorzStn11Hook_27 AT %MX20244.27 : BOOL;
	bArm1HorzStn11Hook_28 AT %MX20244.28 : BOOL;
	bArm1HorzStn11Hook_29 AT %MX20244.29 : BOOL;
	bArm1HorzStn11Hook_30 AT %MX20244.30 : BOOL;
	bArm1HorzStn11Hook_31 AT %MX20244.31 : BOOL;

	bArm1HorzStn12Hook_00 AT %MX20248.0 : BOOL;
	bArm1HorzStn12Hook_01 AT %MX20248.1 : BOOL;
	bArm1HorzStn12Hook_02 AT %MX20248.2 : BOOL;
	bArm1HorzStn12Hook_03 AT %MX20248.3 : BOOL;
	bArm1HorzStn12Hook_04 AT %MX20248.4 : BOOL;
	bArm1HorzStn12Hook_05 AT %MX20248.5 : BOOL;
	bArm1HorzStn12Hook_06 AT %MX20248.6 : BOOL;
	bArm1HorzStn12Hook_07 AT %MX20248.7 : BOOL;
	bArm1HorzStn12Hook_08 AT %MX20248.8 : BOOL;
	bArm1HorzStn12Hook_09 AT %MX20248.9 : BOOL;
	bArm1HorzStn12Hook_10 AT %MX20248.10 : BOOL;
	bArm1HorzStn12Hook_11 AT %MX20248.11 : BOOL;
	bArm1HorzStn12Hook_12 AT %MX20248.12 : BOOL;
	bArm1HorzStn12Hook_13 AT %MX20248.13 : BOOL;
	bArm1HorzStn12Hook_14 AT %MX20248.14 : BOOL;
	bArm1HorzStn12Hook_15 AT %MX20248.15 : BOOL;
	bArm1HorzStn12Hook_16 AT %MX20248.16 : BOOL;
	bArm1HorzStn12Hook_17 AT %MX20248.17 : BOOL;
	bArm1HorzStn12Hook_18 AT %MX20248.18 : BOOL;
	bArm1HorzStn12Hook_19 AT %MX20248.19 : BOOL;
	bArm1HorzStn12Hook_20 AT %MX20248.20 : BOOL;
	bArm1HorzStn12Hook_21 AT %MX20248.21 : BOOL;
	bArm1HorzStn12Hook_22 AT %MX20248.22 : BOOL;
	bArm1HorzStn12Hook_23 AT %MX20248.23 : BOOL;
	bArm1HorzStn12Hook_24 AT %MX20248.24 : BOOL;
	bArm1HorzStn12Hook_25 AT %MX20248.25 : BOOL;
	bArm1HorzStn12Hook_26 AT %MX20248.26 : BOOL;
	bArm1HorzStn12Hook_27 AT %MX20248.27 : BOOL;
	bArm1HorzStn12Hook_28 AT %MX20248.28 : BOOL;
	bArm1HorzStn12Hook_29 AT %MX20248.29 : BOOL;
	bArm1HorzStn12Hook_30 AT %MX20248.30 : BOOL;
	bArm1HorzStn12Hook_31 AT %MX20248.31 : BOOL;


(* xxxxxxxxxxxxxxxxxxxxxxxxxxxxxxxxxxxxxxx Unhook word xxxxxxxxxxxxxxxxxxxxxxxxxxxxxxxxxxxxxxx*)
(*====================== Unhook BOOL LINK with %MX20300-MX20399 ======================*)

	bArm1HorzLD1Unhook_00 AT %MX20352.0 : BOOL;
	bArm1HorzLD1Unhook_01 AT %MX20352.1 : BOOL;
	bArm1HorzLD1Unhook_02 AT %MX20352.2 : BOOL;
	bArm1HorzLD1Unhook_03 AT %MX20352.3 : BOOL;
	bArm1HorzLD1Unhook_04 AT %MX20352.4 : BOOL;
	bArm1HorzLD1Unhook_05 AT %MX20352.5 : BOOL;
	bArm1HorzLD1Unhook_06 AT %MX20352.6 : BOOL;
	bArm1HorzLD1Unhook_07 AT %MX20352.7 : BOOL;
	bArm1HorzLD1Unhook_08 AT %MX20352.8 : BOOL;
	bArm1HorzLD1Unhook_09 AT %MX20352.9 : BOOL;
	bArm1HorzLD1Unhook_10 AT %MX20352.10 : BOOL;
	bArm1HorzLD1Unhook_11 AT %MX20352.11 : BOOL;
	bArm1HorzLD1Unhook_12 AT %MX20352.12 : BOOL;
	bArm1HorzLD1Unhook_13 AT %MX20352.13 : BOOL;
	bArm1HorzLD1Unhook_14 AT %MX20352.14 : BOOL;
	bArm1HorzLD1Unhook_15 AT %MX20352.15 : BOOL;
	bArm1HorzLD1Unhook_16 AT %MX20352.16 : BOOL;
	bArm1HorzLD1Unhook_17 AT %MX20352.17 : BOOL;
	bArm1HorzLD1Unhook_18 AT %MX20352.18 : BOOL;
	bArm1HorzLD1Unhook_19 AT %MX20352.19 : BOOL;
	bArm1HorzLD1Unhook_20 AT %MX20352.20 : BOOL;
	bArm1HorzLD1Unhook_21 AT %MX20352.21 : BOOL;
	bArm1HorzLD1Unhook_22 AT %MX20352.22 : BOOL;
	bArm1HorzLD1Unhook_23 AT %MX20352.23 : BOOL;
	bArm1HorzLD1Unhook_24 AT %MX20352.24 : BOOL;
	bArm1HorzLD1Unhook_25 AT %MX20352.25 : BOOL;
	bArm1HorzLD1Unhook_26 AT %MX20352.26 : BOOL;
	bArm1HorzLD1Unhook_27 AT %MX20352.27 : BOOL;
	bArm1HorzLD1Unhook_28 AT %MX20352.28 : BOOL;
	bArm1HorzLD1Unhook_29 AT %MX20352.29 : BOOL;
	bArm1HorzLD1Unhook_30 AT %MX20352.30 : BOOL;
	bArm1HorzLD1Unhook_31 AT %MX20352.31 : BOOL;

